{region '#Template'}
	{attribute 'Version' := '5.0.0.0'}
	{attribute 'Tags' := '"LCID": "1031", "Text": "AC, Allgemein, AHU, Startprogramm, Aggregat, Kommandierung"'}
	{attribute 'Tags' := '"LCID": "1033", "Text": "AC, General, AHU, Start program, Aggregate, Command"'}
	{attribute 'Using' := '"Type": "Template", "URI": "E_AC_PlantStep01"'}
	{attribute 'Using' := '"Type": "Template", "URI": "E_BA_AC_OpMod01"'}
	{attribute 'Using' := '"Type": "Template", "URI": "FB_BA_AC_OpModAggBinary"'}
	{attribute 'Using' := '"Type": "Template", "URI": "FB_BA_AC_OpModAggMdlt"'}
	{attribute 'Description' := '"LCID": "1031", "Text": "Kommandierung der Anlage FB_BA_AHU_1st_10"'}
	{attribute 'Description' := '"LCID": "1033", "Text": "Commanding the plant FB_BA_AHU_1st_10"'}
{endregion}

FUNCTION_BLOCK FB_BA_AC_PlantCmd_AHU_1st_10 EXTENDS FB_BA_View
VAR_INPUT
	eOpMode						: E_BA_AC_OpMod01;
	stPriorityEn				: ST_BA_PriorityEn;	
	bDmpOuAOpn					: BOOL;		//	Rückmeldung Aussenluftklappe offen		//	Feedback outside air damper open
	bDmpExhAOpn					: BOOL;		//	Rückmeldung Fortluftklappe offen		//	Feedback exhaust air damper open
	bPreRinse					: BOOL;		//	Vorspülen abgeschlossen					//	Prerinse ready
	bMixADmpAvail				: BOOL;		//	Mischluftsystem vorhanden				//	mixing damper system available	
END_VAR
VAR_OUTPUT
	ePltStp						: E_AC_PlantStep01;	//	Stufen des Anlagenstarts	//	Stages of the plant starts	
	stOuADmp					: ST_BA_Binary;
	stExhADmp					: ST_BA_Binary;
	stSuAFan					: ST_BA_Mdlt;
	stExtAFan					: ST_BA_Mdlt;
	stPreHtr					: ST_BA_Binary;
	stCooler					: ST_BA_Binary;
	stErc						: ST_BA_Binary;
	stTempCtrl					: ST_BA_Mdlt;
	bStepCtrlUp					: BOOL;
	bStepCtrlDown				: BOOL;	
END_VAR
VAR_INPUT CONSTANT
	DmpDlyCls					: FB_BA_AV_Op;
	SuAFanDlyOn					: FB_BA_AV_Op;
	ExtAFanDlyOn				: FB_BA_AV_Op;
	TempCtrlDlyOn				: FB_BA_AV_Op;
	PltStp						: FB_BA_MV_Op;
	
	StepCtrlAgg					: FB_BA_StepCtrlAgg16; //	Schrittsteuerung Aggregate // Step control aggregate	
	

	ErcOpMod					: FB_BA_AC_OpModAggBinary;
	ErcStep						: FB_BA_StepBinary;

	PreHtrOpMod					: FB_BA_AC_OpModAggBinary;
	PreHtrStep					: FB_BA_StepBinary;

	OuADmpOpMod					: FB_BA_AC_OpModAggBinary;
	OuADmpStep					: FB_BA_StepBinary;
	
	SuAFanOpMod					: FB_BA_AC_OpModAggMdlt;
	SuAFanStep					: FB_BA_StepMdlt;	

	ExhADmpOpMod				: FB_BA_AC_OpModAggBinary;
	ExhADmpStep					: FB_BA_StepBinary;
	
	ExtAFanOpMod				: FB_BA_AC_OpModAggMdlt;
	ExtAFanStep					: FB_BA_StepMdlt;	

	CoolerOpMod					: FB_BA_AC_OpModAggBinary;
	CoolerStep					: FB_BA_StepBinary;

	TempCtrlOpMod				: FB_BA_AC_OpModAggMdlt;
	TempCtrlStep				: FB_BA_StepMdlt;	
END_VAR
VAR
	stAgg01						: ST_BA_Step;
	stAgg02						: ST_BA_Step;
	stAgg03						: ST_BA_Step;
	stAgg04						: ST_BA_Step;
	stAgg05						: ST_BA_Step;
	stAgg06						: ST_BA_Step;
	stAgg07						: ST_BA_Step;
	stAgg08						: ST_BA_Step;
	stAgg09						: ST_BA_Step;
	stAgg10						: ST_BA_Step;
	stAgg11						: ST_BA_Step;
	stAgg12						: ST_BA_Step;	
	stAgg13						: ST_BA_Step;	
	stAgg14						: ST_BA_Step;	
	stAgg15						: ST_BA_Step;	
	stAgg16						: ST_BA_Step;	
	
	PltStpMMUX					: FB_BA_MMUX_UDI16;	//	Stufen des Anlagenstarts	//	Stages of the plant starts	
END_VAR

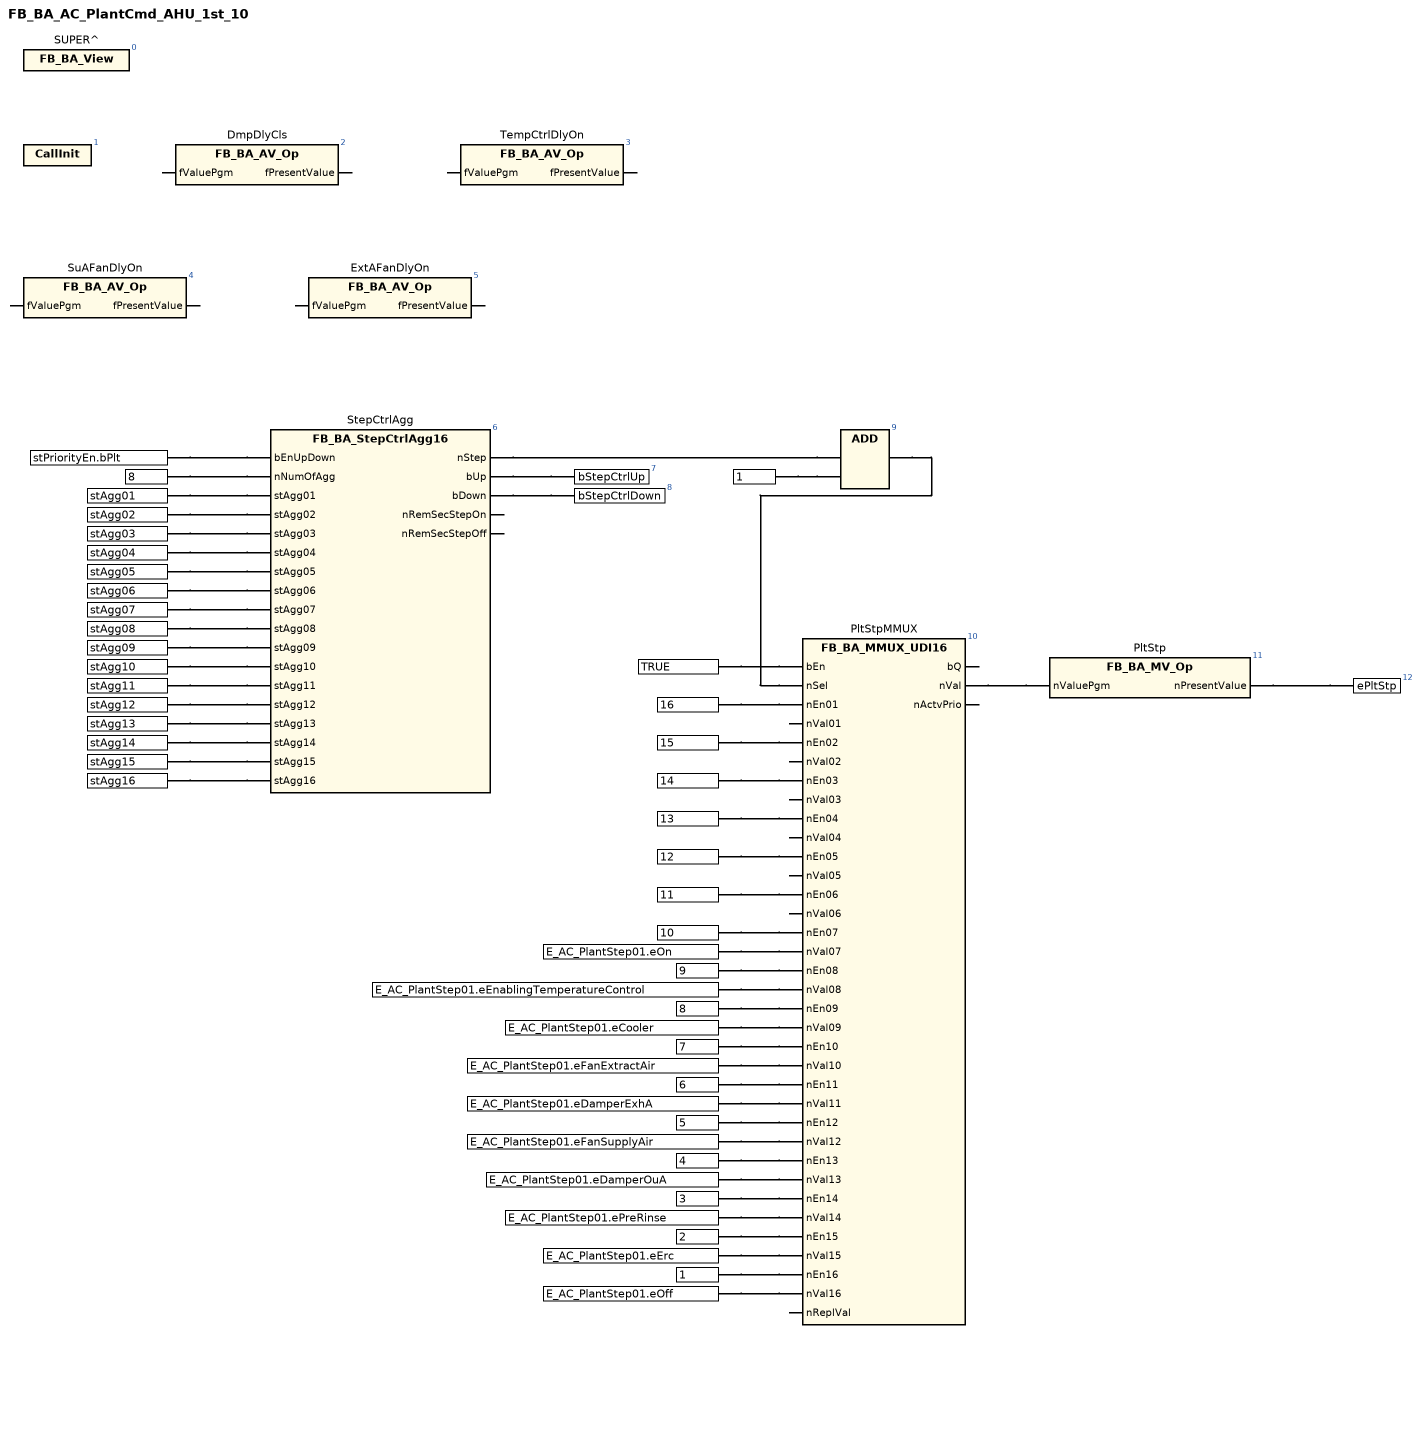
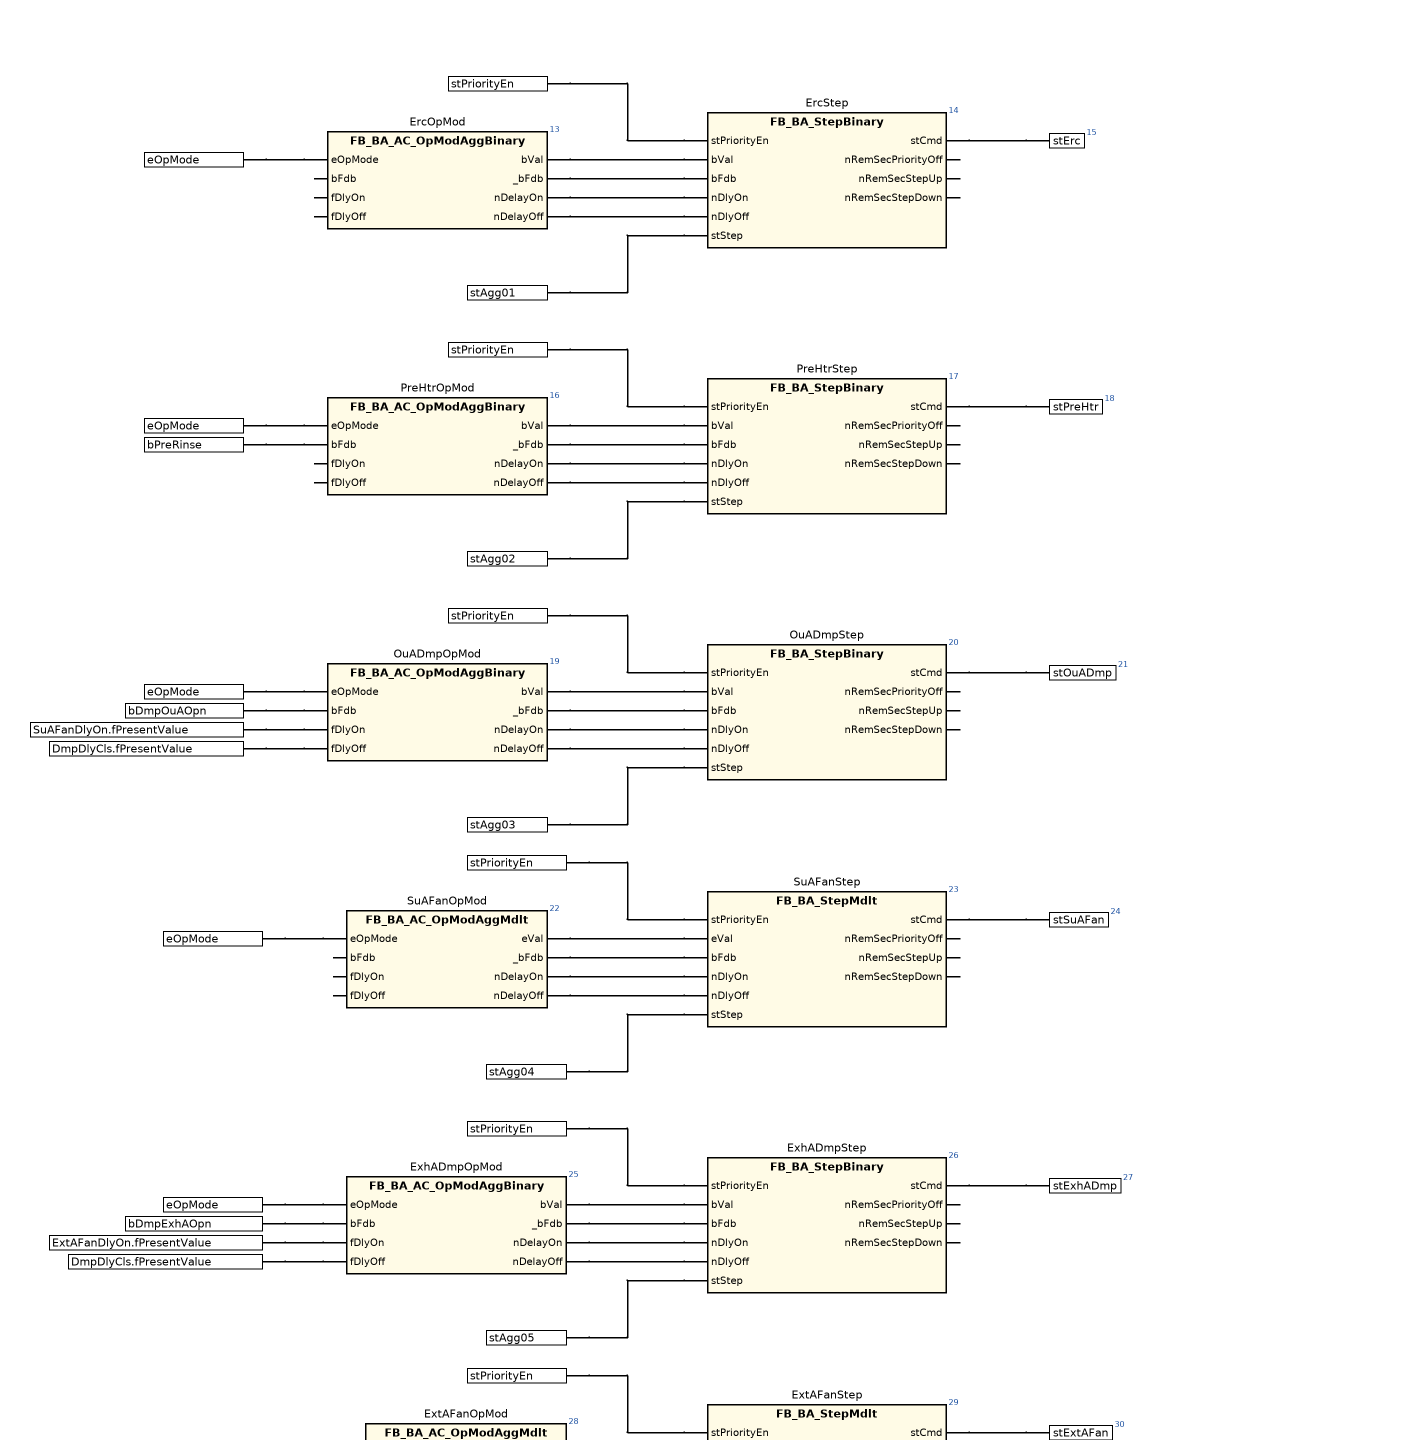
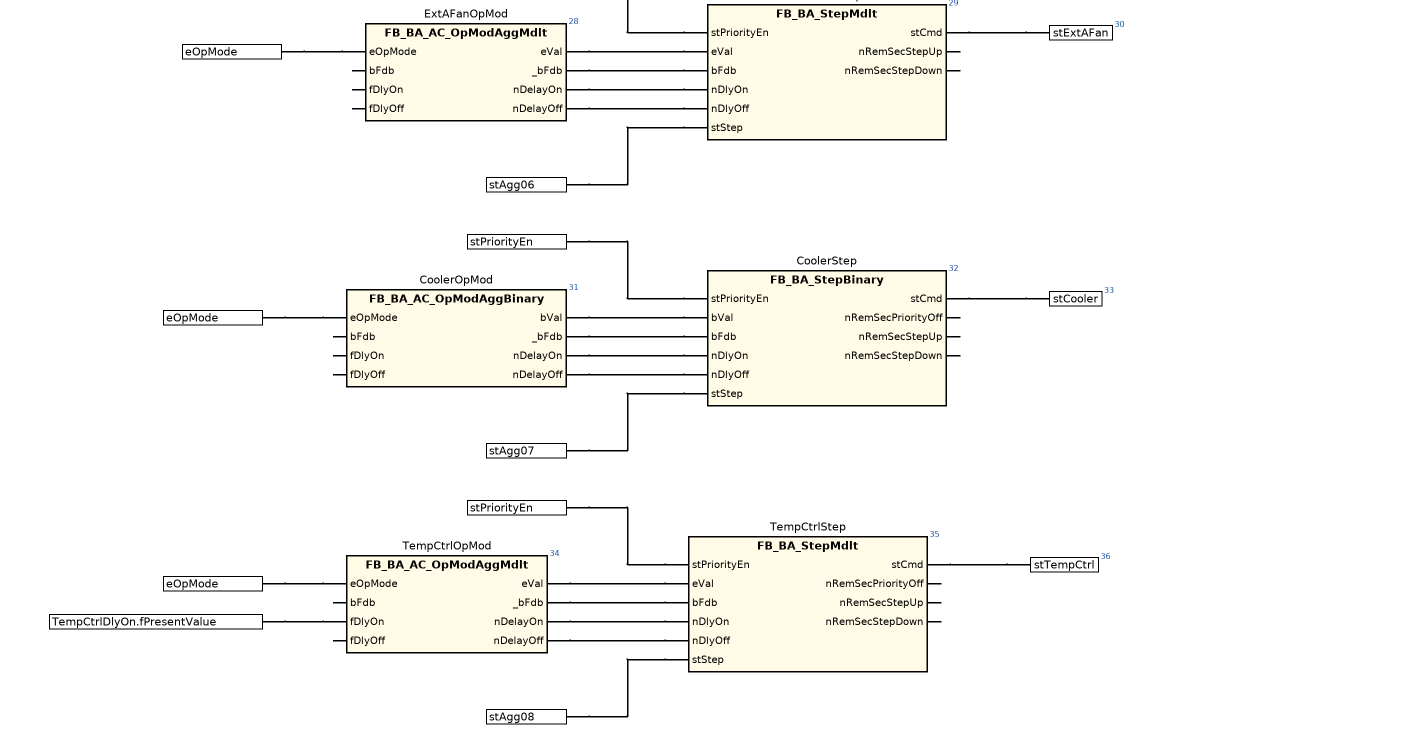
SUPER^(); // FB_BA_View
CallInit();
DmpDlyCls(); // FB_BA_AV_Op
TempCtrlDlyOn(); // FB_BA_AV_Op
SuAFanDlyOn(); // FB_BA_AV_Op
ExtAFanDlyOn(); // FB_BA_AV_Op
StepCtrlAgg(
    bEnUpDown := stPriorityEn.bPlt,
    nNumOfAgg := 8,
    stAgg01 := stAgg01,
    stAgg02 := stAgg02,
    stAgg03 := stAgg03,
    stAgg04 := stAgg04,
    stAgg05 := stAgg05,
    stAgg06 := stAgg06,
    stAgg07 := stAgg07,
    stAgg08 := stAgg08,
    stAgg09 := stAgg09,
    stAgg10 := stAgg10,
    stAgg11 := stAgg11,
    stAgg12 := stAgg12,
    stAgg13 := stAgg13,
    stAgg14 := stAgg14,
    stAgg15 := stAgg15,
    stAgg16 := stAgg16); // FB_BA_StepCtrlAgg16
bStepCtrlUp := StepCtrlAgg.bUp;
bStepCtrlDown := StepCtrlAgg.bDown;
PltStpMMUX(
    bEn := TRUE,
    nSel := StepCtrlAgg.nStep + 1,
    nEn01 := 16,
    nEn02 := 15,
    nEn03 := 14,
    nEn04 := 13,
    nEn05 := 12,
    nEn06 := 11,
    nEn07 := 10,
    nVal07 := E_AC_PlantStep01.eOn,
    nEn08 := 9,
    nVal08 := E_AC_PlantStep01.eEnablingTemperatureControl,
    nEn09 := 8,
    nVal09 := E_AC_PlantStep01.eCooler,
    nEn10 := 7,
    nVal10 := E_AC_PlantStep01.eFanExtractAir,
    nEn11 := 6,
    nVal11 := E_AC_PlantStep01.eDamperExhA,
    nEn12 := 5,
    nVal12 := E_AC_PlantStep01.eFanSupplyAir,
    nEn13 := 4,
    nVal13 := E_AC_PlantStep01.eDamperOuA,
    nEn14 := 3,
    nVal14 := E_AC_PlantStep01.ePreRinse,
    nEn15 := 2,
    nVal15 := E_AC_PlantStep01.eErc,
    nEn16 := 1,
    nVal16 := E_AC_PlantStep01.eOff); // FB_BA_MMUX_UDI16
PltStp(nValuePgm := PltStpMMUX.nVal); // FB_BA_MV_Op
ePltStp := PltStp.nPresentValue;
ErcOpMod(eOpMode := eOpMode); // FB_BA_AC_OpModAggBinary
ErcStep(
    stPriorityEn := stPriorityEn,
    bVal := ErcOpMod.bVal,
    bFdb := ErcOpMod._bFdb,
    nDlyOn := ErcOpMod.nDelayOn,
    nDlyOff := ErcOpMod.nDelayOff,
    stStep := stAgg01); // FB_BA_StepBinary
stErc := ErcStep.stCmd;
PreHtrOpMod(eOpMode := eOpMode, bFdb := bPreRinse); // FB_BA_AC_OpModAggBinary
PreHtrStep(
    stPriorityEn := stPriorityEn,
    bVal := PreHtrOpMod.bVal,
    bFdb := PreHtrOpMod._bFdb,
    nDlyOn := PreHtrOpMod.nDelayOn,
    nDlyOff := PreHtrOpMod.nDelayOff,
    stStep := stAgg02); // FB_BA_StepBinary
stPreHtr := PreHtrStep.stCmd;
OuADmpOpMod(
    eOpMode := eOpMode,
    bFdb := bDmpOuAOpn,
    fDlyOn := SuAFanDlyOn.fPresentValue,
    fDlyOff := DmpDlyCls.fPresentValue); // FB_BA_AC_OpModAggBinary
OuADmpStep(
    stPriorityEn := stPriorityEn,
    bVal := OuADmpOpMod.bVal,
    bFdb := OuADmpOpMod._bFdb,
    nDlyOn := OuADmpOpMod.nDelayOn,
    nDlyOff := OuADmpOpMod.nDelayOff,
    stStep := stAgg03); // FB_BA_StepBinary
stOuADmp := OuADmpStep.stCmd;
SuAFanOpMod(eOpMode := eOpMode); // FB_BA_AC_OpModAggMdlt
SuAFanStep(
    stPriorityEn := stPriorityEn,
    eVal := SuAFanOpMod.eVal,
    bFdb := SuAFanOpMod._bFdb,
    nDlyOn := SuAFanOpMod.nDelayOn,
    nDlyOff := SuAFanOpMod.nDelayOff,
    stStep := stAgg04); // FB_BA_StepMdlt
stSuAFan := SuAFanStep.stCmd;
ExhADmpOpMod(
    eOpMode := eOpMode,
    bFdb := bDmpExhAOpn,
    fDlyOn := ExtAFanDlyOn.fPresentValue,
    fDlyOff := DmpDlyCls.fPresentValue); // FB_BA_AC_OpModAggBinary
ExhADmpStep(
    stPriorityEn := stPriorityEn,
    bVal := ExhADmpOpMod.bVal,
    bFdb := ExhADmpOpMod._bFdb,
    nDlyOn := ExhADmpOpMod.nDelayOn,
    nDlyOff := ExhADmpOpMod.nDelayOff,
    stStep := stAgg05); // FB_BA_StepBinary
stExhADmp := ExhADmpStep.stCmd;
ExtAFanOpMod(eOpMode := eOpMode); // FB_BA_AC_OpModAggMdlt
ExtAFanStep(
    stPriorityEn := stPriorityEn,
    eVal := ExtAFanOpMod.eVal,
    bFdb := ExtAFanOpMod._bFdb,
    nDlyOn := ExtAFanOpMod.nDelayOn,
    nDlyOff := ExtAFanOpMod.nDelayOff,
    stStep := stAgg06); // FB_BA_StepMdlt
stExtAFan := ExtAFanStep.stCmd;
CoolerOpMod(eOpMode := eOpMode); // FB_BA_AC_OpModAggBinary
CoolerStep(
    stPriorityEn := stPriorityEn,
    bVal := CoolerOpMod.bVal,
    bFdb := CoolerOpMod._bFdb,
    nDlyOn := CoolerOpMod.nDelayOn,
    nDlyOff := CoolerOpMod.nDelayOff,
    stStep := stAgg07); // FB_BA_StepBinary
stCooler := CoolerStep.stCmd;
TempCtrlOpMod(eOpMode := eOpMode, fDlyOn := TempCtrlDlyOn.fPresentValue); // FB_BA_AC_OpModAggMdlt
TempCtrlStep(
    stPriorityEn := stPriorityEn,
    eVal := TempCtrlOpMod.eVal,
    bFdb := TempCtrlOpMod._bFdb,
    nDlyOn := TempCtrlOpMod.nDelayOn,
    nDlyOff := TempCtrlOpMod.nDelayOff,
    stStep := stAgg08); // FB_BA_StepMdlt
stTempCtrl := TempCtrlStep.stCmd;

METHOD CallInit
VAR_INPUT
END_VAR
InitErc();
InitPreHtr();

InitOuADmp();
InitSuAFan();

InitExhADmp();
InitExtAFan();

InitCooler();

InitTempCtrl();
END_METHOD

METHOD FB_init : BOOL
VAR_INPUT
	bInitRetains : BOOL; // if TRUE, the retain variables are initialized (warm start / cold start)
	bInCopyCode : BOOL;  // if TRUE, the instance afterwards gets moved into the copy code (online change)
END_VAR
DmpDlyCls.iParent			:= THIS^;
DmpDlyCls.iLabel			:= LblCtl_TimeDelayDampersClose; 	
DmpDlyCls.eUnit				:= E_BA_Unit.eTime_Seconds;  
DmpDlyCls.fValueRm			:= 10;

SuAFanDlyOn.iParent			:= THIS^;
SuAFanDlyOn.iLabel			:= LblCtl_TimeDelaySupplyAirFanOn;   		
SuAFanDlyOn.eUnit			:= E_BA_Unit.eTime_Seconds;  
SuAFanDlyOn.fValueRm		:= 10;

ExtAFanDlyOn.iParent		:= THIS^;
ExtAFanDlyOn.iLabel			:= LblCtl_TimeDelayExtractAirFanOn;   	
ExtAFanDlyOn.eUnit			:= E_BA_Unit.eTime_Seconds;  
ExtAFanDlyOn.fValueRm		:= 10;

TempCtrlDlyOn.iParent		:= THIS^;
TempCtrlDlyOn.iLabel		:= LblCtl_TimeDelayTemperatureSequenceControlOn;   	
TempCtrlDlyOn.eUnit			:= E_BA_Unit.eTime_Seconds;  
TempCtrlDlyOn.fValueRm		:= 5;

PltStp.iParent				:= THIS^;
PltStp.iLabel				:= LblCtl_StagesOfThePlantStartup; 	
PltStp.aStateText[1]		:= txtEvent_Off;
PltStp.aStateText[2]		:= txtEvent_EnergyRecovery;
PltStp.aStateText[3]		:= txtEvent_PreRinse;// or txtEvent_Preheater
PltStp.aStateText[4]		:= txtEvent_DamperOutsideAir;
PltStp.aStateText[5]		:= txtEvent_SupplyAirFan;
PltStp.aStateText[6]		:= txtEvent_DamperExhaustAir;
PltStp.aStateText[7]		:= txtEvent_ExtractAirFan;
PltStp.aStateText[8]		:= txtEvent_Cooler;
PltStp.aStateText[9]		:= txtEvent_Reheater;
PltStp.aStateText[10]		:= txtEvent_MixedAir;
PltStp.aStateText[11]		:= txtEvent_EnableTemperatureControl;
PltStp.aStateText[12]		:= txtEvent_EnableHumidityControl;
PltStp.aStateText[13]		:= txtEvent_On;
END_METHOD

METHOD InitCooler
VAR_INPUT
END_VAR
IF	CoolerOpMod.bInit
THEN	
	CoolerOpMod.bInit := FALSE;
	//////////////////////////////////////////////
	//////////////////////////////////////////////
	//	E_BA_AC_OpMod01.eOff
	CoolerOpMod.arrOpModVal[E_BA_AC_OpMod01.eOff]				:= FALSE;
	CoolerOpMod.arrIgnoreDelayOnVal[E_BA_AC_OpMod01.eOff]		:= TRUE;
	CoolerOpMod.arrIgnoreDelayOffVal[E_BA_AC_OpMod01.eOff]		:= TRUE;
	CoolerOpMod.arrIgnoreFdbVal[E_BA_AC_OpMod01.eOff]			:= TRUE;
	//////////////////////////////////////////////
	//////////////////////////////////////////////
	//	E_BA_AC_OpMod01.eOn
	CoolerOpMod.arrOpModVal[E_BA_AC_OpMod01.eOn]				:= TRUE;
	CoolerOpMod.arrIgnoreDelayOnVal[E_BA_AC_OpMod01.eOn]		:= TRUE;
	CoolerOpMod.arrIgnoreDelayOffVal[E_BA_AC_OpMod01.eOn]		:= TRUE;
	CoolerOpMod.arrIgnoreFdbVal[E_BA_AC_OpMod01.eOn]			:= TRUE;
	//////////////////////////////////////////////
	//////////////////////////////////////////////
	//	E_BA_AC_OpMod01.eEmergency
	CoolerOpMod.arrOpModVal[E_BA_AC_OpMod01.eEmergency]				:= FALSE;
	CoolerOpMod.arrIgnoreDelayOnVal[E_BA_AC_OpMod01.eEmergency]		:= TRUE;
	CoolerOpMod.arrIgnoreDelayOffVal[E_BA_AC_OpMod01.eEmergency]	:= TRUE;
	CoolerOpMod.arrIgnoreFdbVal[E_BA_AC_OpMod01.eEmergency]			:= TRUE;
	//////////////////////////////////////////////
	//////////////////////////////////////////////
	//	E_OpModBA_AC_OpMod01.eFrost
	CoolerOpMod.arrOpModVal[E_BA_AC_OpMod01.eFrost]				:= FALSE;
	CoolerOpMod.arrIgnoreDelayOnVal[E_BA_AC_OpMod01.eFrost]		:= TRUE;
	CoolerOpMod.arrIgnoreDelayOffVal[E_BA_AC_OpMod01.eFrost]	:= TRUE;
	CoolerOpMod.arrIgnoreFdbVal[E_BA_AC_OpMod01.eFrost]			:= TRUE;
	//////////////////////////////////////////////
	//////////////////////////////////////////////
	//	E_BA_AC_OpMod01.eSmokeExtractionProgramm
	CoolerOpMod.arrOpModVal[E_BA_AC_OpMod01.eSmokeExtractionProgram]				:= FALSE;
	CoolerOpMod.arrIgnoreDelayOnVal[E_BA_AC_OpMod01.eSmokeExtractionProgram]		:= TRUE;
	CoolerOpMod.arrIgnoreDelayOffVal[E_BA_AC_OpMod01.eSmokeExtractionProgram]		:= TRUE;
	CoolerOpMod.arrIgnoreFdbVal[E_BA_AC_OpMod01.eSmokeExtractionProgram]			:= TRUE;
	//////////////////////////////////////////////
	//////////////////////////////////////////////
	//	E_BA_AC_OpMod01.eSmokeExtractionSupplyAir
	CoolerOpMod.arrOpModVal[E_BA_AC_OpMod01.eSmokeExtractionSupplyAir]				:= FALSE;
	CoolerOpMod.arrIgnoreDelayOnVal[E_BA_AC_OpMod01.eSmokeExtractionSupplyAir]		:= TRUE;
	CoolerOpMod.arrIgnoreDelayOffVal[E_BA_AC_OpMod01.eSmokeExtractionSupplyAir]		:= TRUE;
	CoolerOpMod.arrIgnoreFdbVal[E_BA_AC_OpMod01.eSmokeExtractionSupplyAir]			:= TRUE;
	//////////////////////////////////////////////
	//////////////////////////////////////////////
	//	E_BA_AC_OpMod01.eSmokeExtractionExhaustAir
	CoolerOpMod.arrOpModVal[E_BA_AC_OpMod01.eSmokeExtractionExhaustAir]				:= FALSE;
	CoolerOpMod.arrIgnoreDelayOnVal[E_BA_AC_OpMod01.eSmokeExtractionExhaustAir]		:= TRUE;
	CoolerOpMod.arrIgnoreDelayOffVal[E_BA_AC_OpMod01.eSmokeExtractionExhaustAir]	:= TRUE;
	CoolerOpMod.arrIgnoreFdbVal[E_BA_AC_OpMod01.eSmokeExtractionExhaustAir]			:= TRUE;
	//////////////////////////////////////////////
	//////////////////////////////////////////////
	//	E_BA_AC_OpMod01.eFire
	CoolerOpMod.arrOpModVal[E_BA_AC_OpMod01.eFire]				:= FALSE;
	CoolerOpMod.arrIgnoreDelayOnVal[E_BA_AC_OpMod01.eFire]		:= TRUE;
	CoolerOpMod.arrIgnoreDelayOffVal[E_BA_AC_OpMod01.eFire]		:= TRUE;
	CoolerOpMod.arrIgnoreFdbVal[E_BA_AC_OpMod01.eFire]			:= TRUE;
	//////////////////////////////////////////////
	//////////////////////////////////////////////
	//	E_BA_AC_OpMod01.eNightCooling
	CoolerOpMod.arrOpModVal[E_BA_AC_OpMod01.eNightCooling]				:= FALSE;
	CoolerOpMod.arrIgnoreDelayOnVal[E_BA_AC_OpMod01.eNightCooling]		:= TRUE;
	CoolerOpMod.arrIgnoreDelayOffVal[E_BA_AC_OpMod01.eNightCooling]		:= TRUE;
	CoolerOpMod.arrIgnoreFdbVal[E_BA_AC_OpMod01.eNightCooling]			:= TRUE;
	//////////////////////////////////////////////
	//////////////////////////////////////////////
	//	E_BA_AC_OpMod01.eCoolDownProtection
	CoolerOpMod.arrOpModVal[E_BA_AC_OpMod01.eCoolDownProtection]				:= FALSE;
	CoolerOpMod.arrIgnoreDelayOnVal[E_BA_AC_OpMod01.eCoolDownProtection]		:= TRUE;
	CoolerOpMod.arrIgnoreDelayOffVal[E_BA_AC_OpMod01.eCoolDownProtection]		:= TRUE;
	CoolerOpMod.arrIgnoreFdbVal[E_BA_AC_OpMod01.eCoolDownProtection]			:= TRUE;
	//////////////////////////////////////////////
	//////////////////////////////////////////////
	//	E_BA_AC_OpMod01.eOverHeatingProtection
	CoolerOpMod.arrOpModVal[E_BA_AC_OpMod01.eOverHeatingProtection]				:= TRUE;
	CoolerOpMod.arrIgnoreDelayOnVal[E_BA_AC_OpMod01.eOverHeatingProtection]		:= TRUE;
	CoolerOpMod.arrIgnoreDelayOffVal[E_BA_AC_OpMod01.eOverHeatingProtection]	:= TRUE;
	CoolerOpMod.arrIgnoreFdbVal[E_BA_AC_OpMod01.eOverHeatingProtection]			:= TRUE;
	//////////////////////////////////////////////
	//////////////////////////////////////////////
	//	E_BA_AC_OpMod01.eAlarm
	CoolerOpMod.arrOpModVal[E_BA_AC_OpMod01.eAlarm]				:= FALSE;
	CoolerOpMod.arrIgnoreDelayOnVal[E_BA_AC_OpMod01.eAlarm]		:= TRUE;
	CoolerOpMod.arrIgnoreDelayOffVal[E_BA_AC_OpMod01.eAlarm]	:= TRUE;
	CoolerOpMod.arrIgnoreFdbVal[E_BA_AC_OpMod01.eAlarm]			:= TRUE;
	//////////////////////////////////////////////
	//////////////////////////////////////////////
	//	E_BA_AC_OpMod01.eForcedVentilation
	CoolerOpMod.arrOpModVal[E_BA_AC_OpMod01.eForcedVentilation]				:= TRUE;
	CoolerOpMod.arrIgnoreDelayOnVal[E_BA_AC_OpMod01.eForcedVentilation]		:= TRUE;
	CoolerOpMod.arrIgnoreDelayOffVal[E_BA_AC_OpMod01.eForcedVentilation]	:= TRUE;
	CoolerOpMod.arrIgnoreFdbVal[E_BA_AC_OpMod01.eForcedVentilation]			:= TRUE;
	//////////////////////////////////////////////
	//////////////////////////////////////////////
	//	E_BA_AC_OpMod01.eCentralSwitchOff
	CoolerOpMod.arrOpModVal[E_BA_AC_OpMod01.eCentralSwitchOff]				:= FALSE;
	CoolerOpMod.arrIgnoreDelayOnVal[E_BA_AC_OpMod01.eCentralSwitchOff]		:= TRUE;
	CoolerOpMod.arrIgnoreDelayOffVal[E_BA_AC_OpMod01.eCentralSwitchOff]		:= TRUE;
	CoolerOpMod.arrIgnoreFdbVal[E_BA_AC_OpMod01.eCentralSwitchOff]			:= TRUE;
	//////////////////////////////////////////////
	//////////////////////////////////////////////
	//	E_BA_AC_OpMod01.eCustomer01
	CoolerOpMod.arrOpModVal[E_BA_AC_OpMod01.eCustomer01]				:= FALSE;
	CoolerOpMod.arrIgnoreDelayOnVal[E_BA_AC_OpMod01.eCustomer01]		:= TRUE;
	CoolerOpMod.arrIgnoreDelayOffVal[E_BA_AC_OpMod01.eCustomer01]		:= TRUE;
	CoolerOpMod.arrIgnoreFdbVal[E_BA_AC_OpMod01.eCustomer01]			:= TRUE;
	//////////////////////////////////////////////
	//////////////////////////////////////////////
	//	E_BA_AC_OpMod01.eCustomer02
	CoolerOpMod.arrOpModVal[E_BA_AC_OpMod01.eCustomer02]				:= FALSE;
	CoolerOpMod.arrIgnoreDelayOnVal[E_BA_AC_OpMod01.eCustomer02]		:= TRUE;
	CoolerOpMod.arrIgnoreDelayOffVal[E_BA_AC_OpMod01.eCustomer02]		:= TRUE;
	CoolerOpMod.arrIgnoreFdbVal[E_BA_AC_OpMod01.eCustomer02]			:= TRUE;
END_IF
END_METHOD

METHOD InitErc
VAR_INPUT
END_VAR
IF	ErcOpMod.bInit
THEN	
	ErcOpMod.bInit := FALSE;
	//////////////////////////////////////////////
	//////////////////////////////////////////////
	//	E_BA_AC_OpMod01.eOff;
	ErcOpMod.arrOpModVal[E_BA_AC_OpMod01.eOff]				:= FALSE;
	ErcOpMod.arrIgnoreDelayOnVal[E_BA_AC_OpMod01.eOff]		:= TRUE;
	ErcOpMod.arrIgnoreDelayOffVal[E_BA_AC_OpMod01.eOff]		:= TRUE;
	ErcOpMod.arrIgnoreFdbVal[E_BA_AC_OpMod01.eOff]			:= TRUE;	
	//////////////////////////////////////////////
	//////////////////////////////////////////////
	//	E_BA_AC_OpMod01.eOn;
	ErcOpMod.arrOpModVal[E_BA_AC_OpMod01.eOn]				:= TRUE;
	ErcOpMod.arrIgnoreDelayOnVal[E_BA_AC_OpMod01.eOn]		:= TRUE;
	ErcOpMod.arrIgnoreDelayOffVal[E_BA_AC_OpMod01.eOn]		:= TRUE;
	ErcOpMod.arrIgnoreFdbVal[E_BA_AC_OpMod01.eOn]			:= TRUE;
	//////////////////////////////////////////////
	//////////////////////////////////////////////
	//	E_BA_AC_OpMod01.eEmergency;
	ErcOpMod.arrOpModVal[E_BA_AC_OpMod01.eEmergency]				:= FALSE;
	ErcOpMod.arrIgnoreDelayOnVal[E_BA_AC_OpMod01.eEmergency]		:= TRUE;
	ErcOpMod.arrIgnoreDelayOffVal[E_BA_AC_OpMod01.eEmergency]		:= TRUE;
	ErcOpMod.arrIgnoreFdbVal[E_BA_AC_OpMod01.eEmergency]			:= TRUE;
	//////////////////////////////////////////////
	//////////////////////////////////////////////
	//	E_BA_AC_OpMod01.eFrost;
	ErcOpMod.arrOpModVal[E_BA_AC_OpMod01.eFrost]				:= FALSE;
	ErcOpMod.arrIgnoreDelayOnVal[E_BA_AC_OpMod01.eFrost]		:= TRUE;
	ErcOpMod.arrIgnoreDelayOffVal[E_BA_AC_OpMod01.eFrost]		:= TRUE;
	ErcOpMod.arrIgnoreFdbVal[E_BA_AC_OpMod01.eFrost]			:= TRUE;
	//////////////////////////////////////////////
	//////////////////////////////////////////////
	//	E_BA_AC_OpMod01.eSmokeExtractionProgramm;
	ErcOpMod.arrOpModVal[E_BA_AC_OpMod01.eSmokeExtractionProgram]				:= FALSE;
	ErcOpMod.arrIgnoreDelayOnVal[E_BA_AC_OpMod01.eSmokeExtractionProgram]		:= TRUE;
	ErcOpMod.arrIgnoreDelayOffVal[E_BA_AC_OpMod01.eSmokeExtractionProgram]		:= TRUE;
	ErcOpMod.arrIgnoreFdbVal[E_BA_AC_OpMod01.eSmokeExtractionProgram]			:= TRUE;
	//////////////////////////////////////////////
	//////////////////////////////////////////////
	//	E_BA_AC_OpMod01.eSmokeExtractionSupplyAir;
	ErcOpMod.arrOpModVal[E_BA_AC_OpMod01.eSmokeExtractionSupplyAir]				:= FALSE;
	ErcOpMod.arrIgnoreDelayOnVal[E_BA_AC_OpMod01.eSmokeExtractionSupplyAir]		:= TRUE;
	ErcOpMod.arrIgnoreDelayOffVal[E_BA_AC_OpMod01.eSmokeExtractionSupplyAir]	:= TRUE;
	ErcOpMod.arrIgnoreFdbVal[E_BA_AC_OpMod01.eSmokeExtractionSupplyAir]			:= TRUE;
	//////////////////////////////////////////////
	//////////////////////////////////////////////
	//	E_BA_AC_OpMod01.eSmokeExtractionExhaustAir;
	ErcOpMod.arrOpModVal[E_BA_AC_OpMod01.eSmokeExtractionExhaustAir]				:= FALSE;
	ErcOpMod.arrIgnoreDelayOnVal[E_BA_AC_OpMod01.eSmokeExtractionExhaustAir]		:= TRUE;
	ErcOpMod.arrIgnoreDelayOffVal[E_BA_AC_OpMod01.eSmokeExtractionExhaustAir]		:= TRUE;
	ErcOpMod.arrIgnoreFdbVal[E_BA_AC_OpMod01.eSmokeExtractionExhaustAir]			:= TRUE;
	//////////////////////////////////////////////
	//////////////////////////////////////////////
	//	E_BA_AC_OpMod01.eFire;
	ErcOpMod.arrOpModVal[E_BA_AC_OpMod01.eFire]				:= FALSE;
	ErcOpMod.arrIgnoreDelayOnVal[E_BA_AC_OpMod01.eFire]		:= TRUE;
	ErcOpMod.arrIgnoreDelayOffVal[E_BA_AC_OpMod01.eFire]	:= TRUE;
	ErcOpMod.arrIgnoreFdbVal[E_BA_AC_OpMod01.eFire]			:= TRUE;
	//////////////////////////////////////////////
	//////////////////////////////////////////////
	//	E_BA_AC_OpMod01.eNightCooling;
	ErcOpMod.arrOpModVal[E_BA_AC_OpMod01.eNightCooling]				:= FALSE;
	ErcOpMod.arrIgnoreDelayOnVal[E_BA_AC_OpMod01.eNightCooling]		:= TRUE;
	ErcOpMod.arrIgnoreDelayOffVal[E_BA_AC_OpMod01.eNightCooling]	:= TRUE;
	ErcOpMod.arrIgnoreFdbVal[E_BA_AC_OpMod01.eNightCooling]			:= TRUE;
	//////////////////////////////////////////////
	//////////////////////////////////////////////
	//	E_BA_AC_OpMod01.eCoolDownProtection;
	ErcOpMod.arrOpModVal[E_BA_AC_OpMod01.eCoolDownProtection]				:= TRUE;
	ErcOpMod.arrIgnoreDelayOnVal[E_BA_AC_OpMod01.eCoolDownProtection]		:= TRUE;
	ErcOpMod.arrIgnoreDelayOffVal[E_BA_AC_OpMod01.eCoolDownProtection]		:= TRUE;
	ErcOpMod.arrIgnoreFdbVal[E_BA_AC_OpMod01.eCoolDownProtection]			:= TRUE;
	//////////////////////////////////////////////
	//////////////////////////////////////////////
	//	E_BA_AC_OpMod01.eOverHeatingProtection;
	ErcOpMod.arrOpModVal[E_BA_AC_OpMod01.eOverHeatingProtection]			:= TRUE;
	ErcOpMod.arrIgnoreDelayOnVal[E_BA_AC_OpMod01.eOverHeatingProtection]	:= TRUE;
	ErcOpMod.arrIgnoreDelayOffVal[E_BA_AC_OpMod01.eOverHeatingProtection]	:= TRUE;
	ErcOpMod.arrIgnoreFdbVal[E_BA_AC_OpMod01.eOverHeatingProtection]		:= TRUE;
	//////////////////////////////////////////////
	//////////////////////////////////////////////
	//	E_BA_AC_OpMod01.eAlarm;
	ErcOpMod.arrOpModVal[E_BA_AC_OpMod01.eAlarm]				:= FALSE;
	ErcOpMod.arrIgnoreDelayOnVal[E_BA_AC_OpMod01.eAlarm]		:= TRUE;
	ErcOpMod.arrIgnoreDelayOffVal[E_BA_AC_OpMod01.eAlarm]		:= TRUE;
	ErcOpMod.arrIgnoreFdbVal[E_BA_AC_OpMod01.eAlarm]			:= TRUE;
	//////////////////////////////////////////////
	//////////////////////////////////////////////
	//	E_BA_AC_OpMod01.eForcedVentilation;
	ErcOpMod.arrOpModVal[E_BA_AC_OpMod01.eForcedVentilation]				:= TRUE;
	ErcOpMod.arrIgnoreDelayOnVal[E_BA_AC_OpMod01.eForcedVentilation]		:= TRUE;
	ErcOpMod.arrIgnoreDelayOffVal[E_BA_AC_OpMod01.eForcedVentilation]		:= TRUE;
	ErcOpMod.arrIgnoreFdbVal[E_BA_AC_OpMod01.eForcedVentilation]			:= TRUE;
	//////////////////////////////////////////////
	//////////////////////////////////////////////
	//	E_BA_AC_OpMod01.eCentralSwitchOff;
	ErcOpMod.arrOpModVal[E_BA_AC_OpMod01.eCentralSwitchOff]				:= FALSE;
	ErcOpMod.arrIgnoreDelayOnVal[E_BA_AC_OpMod01.eCentralSwitchOff]		:= TRUE;
	ErcOpMod.arrIgnoreDelayOffVal[E_BA_AC_OpMod01.eCentralSwitchOff]	:= TRUE;
	ErcOpMod.arrIgnoreFdbVal[E_BA_AC_OpMod01.eCentralSwitchOff]			:= TRUE;
	//////////////////////////////////////////////
	//////////////////////////////////////////////
	//	E_BA_AC_OpMod01.eCustomer01;
	ErcOpMod.arrOpModVal[E_BA_AC_OpMod01.eCustomer01]				:= FALSE;
	ErcOpMod.arrIgnoreDelayOnVal[E_BA_AC_OpMod01.eCustomer01]		:= TRUE;
	ErcOpMod.arrIgnoreDelayOffVal[E_BA_AC_OpMod01.eCustomer01]		:= TRUE;
	ErcOpMod.arrIgnoreFdbVal[E_BA_AC_OpMod01.eCustomer01]			:= TRUE;
	//////////////////////////////////////////////
	//////////////////////////////////////////////
	//	E_BA_AC_OpMod01.eCustomer02;
	ErcOpMod.arrOpModVal[E_BA_AC_OpMod01.eCustomer02]				:= FALSE;
	ErcOpMod.arrIgnoreDelayOnVal[E_BA_AC_OpMod01.eCustomer02]		:= TRUE;
	ErcOpMod.arrIgnoreDelayOffVal[E_BA_AC_OpMod01.eCustomer02]		:= TRUE;
	ErcOpMod.arrIgnoreFdbVal[E_BA_AC_OpMod01.eCustomer02]			:= TRUE;
END_IF
END_METHOD

METHOD InitExhADmp
VAR_INPUT
END_VAR
IF	ExhADmpOpMod.bInit
THEN	
	ExhADmpOpMod.bInit := FALSE;
	//////////////////////////////////////////////
	//////////////////////////////////////////////
	//	E_BA_AC_OpMod01.eOff
	ExhADmpOpMod.arrOpModVal[E_BA_AC_OpMod01.eOff]				:= FALSE;
	ExhADmpOpMod.arrIgnoreDelayOnVal[E_BA_AC_OpMod01.eOff]		:= TRUE;
	ExhADmpOpMod.arrIgnoreDelayOffVal[E_BA_AC_OpMod01.eOff]		:= FALSE;
	ExhADmpOpMod.arrIgnoreFdbVal[E_BA_AC_OpMod01.eOff]			:= TRUE;
	//////////////////////////////////////////////
	//////////////////////////////////////////////
	//	E_BA_AC_OpMod01.eOn;
	ExhADmpOpMod.arrOpModVal[E_BA_AC_OpMod01.eOn]				:= TRUE;
	ExhADmpOpMod.arrIgnoreDelayOnVal[E_BA_AC_OpMod01.eOn]		:= TRUE;
	ExhADmpOpMod.arrIgnoreDelayOffVal[E_BA_AC_OpMod01.eOn]		:= TRUE;
	ExhADmpOpMod.arrIgnoreFdbVal[E_BA_AC_OpMod01.eOn]			:= FALSE;
	//////////////////////////////////////////////
	//////////////////////////////////////////////
	//	E_BA_AC_OpMod01.eEmergency;
	ExhADmpOpMod.arrOpModVal[E_BA_AC_OpMod01.eEmergency]				:= FALSE;
	ExhADmpOpMod.arrIgnoreDelayOnVal[E_BA_AC_OpMod01.eEmergency]		:= TRUE;
	ExhADmpOpMod.arrIgnoreDelayOffVal[E_BA_AC_OpMod01.eEmergency]		:= TRUE;
	ExhADmpOpMod.arrIgnoreFdbVal[E_BA_AC_OpMod01.eEmergency]			:= TRUE;
	//////////////////////////////////////////////
	//////////////////////////////////////////////
	//	E_BA_AC_OpMod01.eFrost;
	ExhADmpOpMod.arrOpModVal[E_BA_AC_OpMod01.eFrost]				:= FALSE;
	ExhADmpOpMod.arrIgnoreDelayOnVal[E_BA_AC_OpMod01.eFrost]		:= TRUE;
	ExhADmpOpMod.arrIgnoreDelayOffVal[E_BA_AC_OpMod01.eFrost]		:= FALSE;
	ExhADmpOpMod.arrIgnoreFdbVal[E_BA_AC_OpMod01.eFrost]			:= TRUE;
	//////////////////////////////////////////////
	//////////////////////////////////////////////
	//	E_BA_AC_OpMod01.eSmokeExtractionProgramm;
	ExhADmpOpMod.arrOpModVal[E_BA_AC_OpMod01.eSmokeExtractionProgram]				:= TRUE;
	ExhADmpOpMod.arrIgnoreDelayOnVal[E_BA_AC_OpMod01.eSmokeExtractionProgram]		:= TRUE;
	ExhADmpOpMod.arrIgnoreDelayOffVal[E_BA_AC_OpMod01.eSmokeExtractionProgram]		:= TRUE;
	ExhADmpOpMod.arrIgnoreFdbVal[E_BA_AC_OpMod01.eSmokeExtractionProgram]			:= TRUE;
	//////////////////////////////////////////////
	//////////////////////////////////////////////
	//	E_BA_AC_OpMod01.eSmokeExtractionSupplyAir;
	ExhADmpOpMod.arrOpModVal[E_BA_AC_OpMod01.eSmokeExtractionSupplyAir]				:= FALSE;
	ExhADmpOpMod.arrIgnoreDelayOnVal[E_BA_AC_OpMod01.eSmokeExtractionSupplyAir]		:= TRUE;
	ExhADmpOpMod.arrIgnoreDelayOffVal[E_BA_AC_OpMod01.eSmokeExtractionSupplyAir]	:= FALSE;
	ExhADmpOpMod.arrIgnoreFdbVal[E_BA_AC_OpMod01.eSmokeExtractionSupplyAir]			:= TRUE;
	//////////////////////////////////////////////
	//////////////////////////////////////////////
	//	E_BA_AC_OpMod01.eSmokeExtractionExhaustAir;
	ExhADmpOpMod.arrOpModVal[E_BA_AC_OpMod01.eSmokeExtractionExhaustAir]				:= TRUE;
	ExhADmpOpMod.arrIgnoreDelayOnVal[E_BA_AC_OpMod01.eSmokeExtractionExhaustAir]		:= TRUE;
	ExhADmpOpMod.arrIgnoreDelayOffVal[E_BA_AC_OpMod01.eSmokeExtractionExhaustAir]		:= TRUE;
	ExhADmpOpMod.arrIgnoreFdbVal[E_BA_AC_OpMod01.eSmokeExtractionExhaustAir]			:= TRUE;
	//////////////////////////////////////////////
	//////////////////////////////////////////////
	//	E_BA_AC_OpMod01.eFire;
	ExhADmpOpMod.arrOpModVal[E_BA_AC_OpMod01.eFire]				:= FALSE;
	ExhADmpOpMod.arrIgnoreDelayOnVal[E_BA_AC_OpMod01.eFire]		:= TRUE;
	ExhADmpOpMod.arrIgnoreDelayOffVal[E_BA_AC_OpMod01.eFire]	:= TRUE;
	ExhADmpOpMod.arrIgnoreFdbVal[E_BA_AC_OpMod01.eFire]			:= TRUE;
	//////////////////////////////////////////////
	//////////////////////////////////////////////
	//	E_BA_AC_OpMod01.eNightCooling;
	ExhADmpOpMod.arrOpModVal[E_BA_AC_OpMod01.eNightCooling]				:= TRUE;
	ExhADmpOpMod.arrIgnoreDelayOnVal[E_BA_AC_OpMod01.eNightCooling]		:= TRUE;
	ExhADmpOpMod.arrIgnoreDelayOffVal[E_BA_AC_OpMod01.eNightCooling]	:= TRUE;
	ExhADmpOpMod.arrIgnoreFdbVal[E_BA_AC_OpMod01.eNightCooling]			:= FALSE;
	//////////////////////////////////////////////
	//////////////////////////////////////////////
	//	E_BA_AC_OpMod01.eCoolDownProtection;
	ExhADmpOpMod.arrOpModVal[E_BA_AC_OpMod01.eCoolDownProtection]				:= TRUE;
	ExhADmpOpMod.arrIgnoreDelayOnVal[E_BA_AC_OpMod01.eCoolDownProtection]		:= TRUE;
	ExhADmpOpMod.arrIgnoreDelayOffVal[E_BA_AC_OpMod01.eCoolDownProtection]		:= TRUE;
	ExhADmpOpMod.arrIgnoreFdbVal[E_BA_AC_OpMod01.eCoolDownProtection]			:= FALSE;
	//////////////////////////////////////////////
	//////////////////////////////////////////////
	//	E_BA_AC_OpMod01.eOverHeatingProtection;
	ExhADmpOpMod.arrOpModVal[E_BA_AC_OpMod01.eOverHeatingProtection]				:= TRUE;
	ExhADmpOpMod.arrIgnoreDelayOnVal[E_BA_AC_OpMod01.eOverHeatingProtection]		:= TRUE;
	ExhADmpOpMod.arrIgnoreDelayOffVal[E_BA_AC_OpMod01.eOverHeatingProtection]		:= TRUE;
	ExhADmpOpMod.arrIgnoreFdbVal[E_BA_AC_OpMod01.eOverHeatingProtection]			:= FALSE;
	//////////////////////////////////////////////
	//////////////////////////////////////////////
	//	E_BA_AC_OpMod01.eAlarm;
	ExhADmpOpMod.arrOpModVal[E_BA_AC_OpMod01.eAlarm]				:= FALSE;
	ExhADmpOpMod.arrIgnoreDelayOnVal[E_BA_AC_OpMod01.eAlarm]		:= TRUE;
	ExhADmpOpMod.arrIgnoreDelayOffVal[E_BA_AC_OpMod01.eAlarm]		:= FALSE;
	ExhADmpOpMod.arrIgnoreFdbVal[E_BA_AC_OpMod01.eAlarm]			:= TRUE;
	//////////////////////////////////////////////
	//////////////////////////////////////////////
	//	E_BA_AC_OpMod01.eForcedVentilation;
	ExhADmpOpMod.arrOpModVal[E_BA_AC_OpMod01.eForcedVentilation]				:= TRUE;
	ExhADmpOpMod.arrIgnoreDelayOnVal[E_BA_AC_OpMod01.eForcedVentilation]		:= TRUE;
	ExhADmpOpMod.arrIgnoreDelayOffVal[E_BA_AC_OpMod01.eForcedVentilation]		:= TRUE;
	ExhADmpOpMod.arrIgnoreFdbVal[E_BA_AC_OpMod01.eForcedVentilation]			:= FALSE;
	//////////////////////////////////////////////
	//////////////////////////////////////////////
	//	E_BA_AC_OpMod01.eCentralSwitchOff;
	ExhADmpOpMod.arrOpModVal[E_BA_AC_OpMod01.eCentralSwitchOff]				:= FALSE;
	ExhADmpOpMod.arrIgnoreDelayOnVal[E_BA_AC_OpMod01.eCentralSwitchOff]		:= TRUE;
	ExhADmpOpMod.arrIgnoreDelayOffVal[E_BA_AC_OpMod01.eCentralSwitchOff]	:= FALSE;
	ExhADmpOpMod.arrIgnoreFdbVal[E_BA_AC_OpMod01.eCentralSwitchOff]			:= TRUE;
	//////////////////////////////////////////////
	//////////////////////////////////////////////
	//	E_BA_AC_OpMod01.eCustomer01;
	ExhADmpOpMod.arrOpModVal[E_BA_AC_OpMod01.eCustomer01]				:= FALSE;
	ExhADmpOpMod.arrIgnoreDelayOnVal[E_BA_AC_OpMod01.eCustomer01]		:= TRUE;
	ExhADmpOpMod.arrIgnoreDelayOffVal[E_BA_AC_OpMod01.eCustomer01]		:= FALSE;
	ExhADmpOpMod.arrIgnoreFdbVal[E_BA_AC_OpMod01.eCustomer01]			:= TRUE;
	//////////////////////////////////////////////
	//////////////////////////////////////////////
	//	E_BA_AC_OpMod01.eCustomer02;
	ExhADmpOpMod.arrOpModVal[E_BA_AC_OpMod01.eCustomer02]				:= FALSE;
	ExhADmpOpMod.arrIgnoreDelayOnVal[E_BA_AC_OpMod01.eCustomer02]		:= TRUE;
	ExhADmpOpMod.arrIgnoreDelayOffVal[E_BA_AC_OpMod01.eCustomer02]		:= FALSE;
	ExhADmpOpMod.arrIgnoreFdbVal[E_BA_AC_OpMod01.eCustomer02]			:= TRUE;
END_IF
END_METHOD

METHOD InitExtAFan
VAR_INPUT
END_VAR
IF	ExtAFanOpMod.bInit
THEN	
	ExtAFanOpMod.bInit := FALSE;
	//////////////////////////////////////////////
	//////////////////////////////////////////////
	//	E_BA_AC_OpMod01.eOff;
	ExtAFanOpMod.arrOpModVal[E_BA_AC_OpMod01.eOff]				:= E_BA_Mdlt.eOff;
	ExtAFanOpMod.arrIgnoreDelayOnVal[E_BA_AC_OpMod01.eOff]		:= TRUE;
	ExtAFanOpMod.arrIgnoreDelayOffVal[E_BA_AC_OpMod01.eOff]		:= TRUE;
	ExtAFanOpMod.arrIgnoreFdbVal[E_BA_AC_OpMod01.eOff]			:= TRUE;
	//////////////////////////////////////////////
	//////////////////////////////////////////////
	//	E_BA_AC_OpMod01.eOn;
	ExtAFanOpMod.arrOpModVal[E_BA_AC_OpMod01.eOn]				:= E_BA_Mdlt.eOn;
	ExtAFanOpMod.arrIgnoreDelayOnVal[E_BA_AC_OpMod01.eOn]		:= FALSE;
	ExtAFanOpMod.arrIgnoreDelayOffVal[E_BA_AC_OpMod01.eOn]		:= TRUE;
	ExtAFanOpMod.arrIgnoreFdbVal[E_BA_AC_OpMod01.eOn]			:= TRUE;
	//////////////////////////////////////////////
	//////////////////////////////////////////////
	//	E_BA_AC_OpMod01.eEmergency;
	ExtAFanOpMod.arrOpModVal[E_BA_AC_OpMod01.eEmergency]				:= E_BA_Mdlt.eOff;
	ExtAFanOpMod.arrIgnoreDelayOnVal[E_BA_AC_OpMod01.eEmergency]		:= TRUE;
	ExtAFanOpMod.arrIgnoreDelayOffVal[E_BA_AC_OpMod01.eEmergency]		:= TRUE;
	ExtAFanOpMod.arrIgnoreFdbVal[E_BA_AC_OpMod01.eEmergency]			:= TRUE;
	//////////////////////////////////////////////
	//////////////////////////////////////////////
	//	E_BA_AC_OpMod01.eFrost;
	ExtAFanOpMod.arrOpModVal[E_BA_AC_OpMod01.eFrost]				:= E_BA_Mdlt.eOff;
	ExtAFanOpMod.arrIgnoreDelayOnVal[E_BA_AC_OpMod01.eFrost]		:= TRUE;
	ExtAFanOpMod.arrIgnoreDelayOffVal[E_BA_AC_OpMod01.eFrost]		:= TRUE;
	ExtAFanOpMod.arrIgnoreFdbVal[E_BA_AC_OpMod01.eFrost]			:= TRUE;
	//////////////////////////////////////////////
	//////////////////////////////////////////////
	//	E_BA_AC_OpMod01.eSmokeExtractionProgramm;
	ExtAFanOpMod.arrOpModVal[E_BA_AC_OpMod01.eSmokeExtractionProgram]				:= E_BA_Mdlt.eOn;
	ExtAFanOpMod.arrIgnoreDelayOnVal[E_BA_AC_OpMod01.eSmokeExtractionProgram]		:= TRUE;
	ExtAFanOpMod.arrIgnoreDelayOffVal[E_BA_AC_OpMod01.eSmokeExtractionProgram]		:= TRUE;
	ExtAFanOpMod.arrIgnoreFdbVal[E_BA_AC_OpMod01.eSmokeExtractionProgram]			:= TRUE;
	//////////////////////////////////////////////
	//////////////////////////////////////////////
	//	E_BA_AC_OpMod01.eSmokeExtractionSupplyAir;
	ExtAFanOpMod.arrOpModVal[E_BA_AC_OpMod01.eSmokeExtractionSupplyAir]				:= E_BA_Mdlt.eOff;
	ExtAFanOpMod.arrIgnoreDelayOnVal[E_BA_AC_OpMod01.eSmokeExtractionSupplyAir]		:= TRUE;
	ExtAFanOpMod.arrIgnoreDelayOffVal[E_BA_AC_OpMod01.eSmokeExtractionSupplyAir]	:= TRUE;
	ExtAFanOpMod.arrIgnoreFdbVal[E_BA_AC_OpMod01.eSmokeExtractionSupplyAir]			:= TRUE;
	//////////////////////////////////////////////
	//////////////////////////////////////////////
	//	E_BA_AC_OpMod01.eSmokeExtractionExhaustAir;
	ExtAFanOpMod.arrOpModVal[E_BA_AC_OpMod01.eSmokeExtractionExhaustAir]				:= E_BA_Mdlt.eOn;
	ExtAFanOpMod.arrIgnoreDelayOnVal[E_BA_AC_OpMod01.eSmokeExtractionExhaustAir]		:= TRUE;
	ExtAFanOpMod.arrIgnoreDelayOffVal[E_BA_AC_OpMod01.eSmokeExtractionExhaustAir]		:= TRUE;
	ExtAFanOpMod.arrIgnoreFdbVal[E_BA_AC_OpMod01.eSmokeExtractionExhaustAir]			:= TRUE;
	//////////////////////////////////////////////
	//////////////////////////////////////////////
	//	E_BA_AC_OpMod01.eFire;
	ExtAFanOpMod.arrOpModVal[E_BA_AC_OpMod01.eFire]				:= E_BA_Mdlt.eOff;
	ExtAFanOpMod.arrIgnoreDelayOnVal[E_BA_AC_OpMod01.eFire]		:= TRUE;
	ExtAFanOpMod.arrIgnoreDelayOffVal[E_BA_AC_OpMod01.eFire]	:= TRUE;
	ExtAFanOpMod.arrIgnoreFdbVal[E_BA_AC_OpMod01.eFire]			:= TRUE;
	//////////////////////////////////////////////
	//////////////////////////////////////////////
	//	E_BA_AC_OpMod01.eNightCooling;
	ExtAFanOpMod.arrOpModVal[E_BA_AC_OpMod01.eNightCooling]				:= E_BA_Mdlt.eOn;
	ExtAFanOpMod.arrIgnoreDelayOnVal[E_BA_AC_OpMod01.eNightCooling]		:= TRUE;
	ExtAFanOpMod.arrIgnoreDelayOffVal[E_BA_AC_OpMod01.eNightCooling]	:= TRUE;
	ExtAFanOpMod.arrIgnoreFdbVal[E_BA_AC_OpMod01.eNightCooling]			:= TRUE;
	//////////////////////////////////////////////
	//////////////////////////////////////////////
	//	E_BA_AC_OpMod01.eCoolDownProtection;
	ExtAFanOpMod.arrOpModVal[E_BA_AC_OpMod01.eCoolDownProtection]				:= E_BA_Mdlt.eOn;
	ExtAFanOpMod.arrIgnoreDelayOnVal[E_BA_AC_OpMod01.eCoolDownProtection]		:= TRUE;
	ExtAFanOpMod.arrIgnoreDelayOffVal[E_BA_AC_OpMod01.eCoolDownProtection]		:= TRUE;
	ExtAFanOpMod.arrIgnoreFdbVal[E_BA_AC_OpMod01.eCoolDownProtection]			:= TRUE;
	//////////////////////////////////////////////
	//////////////////////////////////////////////
	//	E_BA_AC_OpMod01.eOverHeatingProtection;
	ExtAFanOpMod.arrOpModVal[E_BA_AC_OpMod01.eOverHeatingProtection]				:= E_BA_Mdlt.eOn;
	ExtAFanOpMod.arrIgnoreDelayOnVal[E_BA_AC_OpMod01.eOverHeatingProtection]		:= TRUE;
	ExtAFanOpMod.arrIgnoreDelayOffVal[E_BA_AC_OpMod01.eOverHeatingProtection]		:= TRUE;
	ExtAFanOpMod.arrIgnoreFdbVal[E_BA_AC_OpMod01.eOverHeatingProtection]			:= TRUE;
	//////////////////////////////////////////////
	//////////////////////////////////////////////
	//	E_BA_AC_OpMod01.eAlarm;
	ExtAFanOpMod.arrOpModVal[E_BA_AC_OpMod01.eAlarm]				:= E_BA_Mdlt.eOff;
	ExtAFanOpMod.arrIgnoreDelayOnVal[E_BA_AC_OpMod01.eAlarm]		:= TRUE;
	ExtAFanOpMod.arrIgnoreDelayOffVal[E_BA_AC_OpMod01.eAlarm]		:= TRUE;
	ExtAFanOpMod.arrIgnoreFdbVal[E_BA_AC_OpMod01.eAlarm]			:= TRUE;
	//////////////////////////////////////////////
	//////////////////////////////////////////////
	//	E_BA_AC_OpMod01.eForcedVentilation;
	ExtAFanOpMod.arrOpModVal[E_BA_AC_OpMod01.eForcedVentilation]				:= E_BA_Mdlt.eOn;
	ExtAFanOpMod.arrIgnoreDelayOnVal[E_BA_AC_OpMod01.eForcedVentilation]		:= TRUE;
	ExtAFanOpMod.arrIgnoreDelayOffVal[E_BA_AC_OpMod01.eForcedVentilation]		:= TRUE;
	ExtAFanOpMod.arrIgnoreFdbVal[E_BA_AC_OpMod01.eForcedVentilation]			:= TRUE;
	//////////////////////////////////////////////
	//////////////////////////////////////////////
	//	E_BA_AC_OpMod01.eCentralSwitchOff;
	ExtAFanOpMod.arrOpModVal[E_BA_AC_OpMod01.eCentralSwitchOff]				:= E_BA_Mdlt.eOff;
	ExtAFanOpMod.arrIgnoreDelayOnVal[E_BA_AC_OpMod01.eCentralSwitchOff]		:= TRUE;
	ExtAFanOpMod.arrIgnoreDelayOffVal[E_BA_AC_OpMod01.eCentralSwitchOff]	:= TRUE;
	ExtAFanOpMod.arrIgnoreFdbVal[E_BA_AC_OpMod01.eCentralSwitchOff]			:= TRUE;
	//////////////////////////////////////////////
	//////////////////////////////////////////////
	//	E_BA_AC_OpMod01.eCustomer01;
	ExtAFanOpMod.arrOpModVal[E_BA_AC_OpMod01.eCustomer01]				:= E_BA_Mdlt.eOff;
	ExtAFanOpMod.arrIgnoreDelayOnVal[E_BA_AC_OpMod01.eCustomer01]		:= TRUE;
	ExtAFanOpMod.arrIgnoreDelayOffVal[E_BA_AC_OpMod01.eCustomer01]		:= TRUE;
	ExtAFanOpMod.arrIgnoreFdbVal[E_BA_AC_OpMod01.eCustomer01]			:= TRUE;
	//////////////////////////////////////////////
	//////////////////////////////////////////////
	//	E_BA_AC_OpMod01.eCustomer02;
	ExtAFanOpMod.arrOpModVal[E_BA_AC_OpMod01.eCustomer02]				:= E_BA_Mdlt.eOff;
	ExtAFanOpMod.arrIgnoreDelayOnVal[E_BA_AC_OpMod01.eCustomer02]		:= TRUE;
	ExtAFanOpMod.arrIgnoreDelayOffVal[E_BA_AC_OpMod01.eCustomer02]		:= TRUE;
	ExtAFanOpMod.arrIgnoreFdbVal[E_BA_AC_OpMod01.eCustomer02]			:= TRUE;
END_IF
END_METHOD

METHOD InitOuADmp
VAR_INPUT
END_VAR
IF	OuADmpOpMod.bInit
THEN	
	OuADmpOpMod.bInit := FALSE;
	//////////////////////////////////////////////
	//////////////////////////////////////////////
	//	E_BA_AC_OpMod01.eOff;
	OuADmpOpMod.arrOpModVal[E_BA_AC_OpMod01.eOff]				:= FALSE;
	OuADmpOpMod.arrIgnoreDelayOnVal[E_BA_AC_OpMod01.eOff]		:= TRUE;
	OuADmpOpMod.arrIgnoreDelayOffVal[E_BA_AC_OpMod01.eOff]		:= FALSE;
	OuADmpOpMod.arrIgnoreFdbVal[E_BA_AC_OpMod01.eOff]			:= TRUE;
	//////////////////////////////////////////////
	//////////////////////////////////////////////
	//	E_BA_AC_OpMod01.eOn;
	OuADmpOpMod.arrOpModVal[E_BA_AC_OpMod01.eOn]				:= TRUE;
	OuADmpOpMod.arrIgnoreDelayOnVal[E_BA_AC_OpMod01.eOn]		:= TRUE;
	OuADmpOpMod.arrIgnoreDelayOffVal[E_BA_AC_OpMod01.eOn]	:= TRUE;
	OuADmpOpMod.arrIgnoreFdbVal[E_BA_AC_OpMod01.eOn]			:= FALSE;
	//////////////////////////////////////////////
	//////////////////////////////////////////////	
	//	E_BA_AC_OpMod01.eEmergency;
	OuADmpOpMod.arrOpModVal[E_BA_AC_OpMod01.eEmergency]				:= FALSE;
	OuADmpOpMod.arrIgnoreDelayOnVal[E_BA_AC_OpMod01.eEmergency]		:= TRUE;
	OuADmpOpMod.arrIgnoreDelayOffVal[E_BA_AC_OpMod01.eEmergency]		:= FALSE;
	OuADmpOpMod.arrIgnoreFdbVal[E_BA_AC_OpMod01.eEmergency]			:= TRUE;
	//////////////////////////////////////////////
	//////////////////////////////////////////////
	//	E_BA_AC_OpMod01.eFrost;
	OuADmpOpMod.arrOpModVal[E_BA_AC_OpMod01.eFrost]				:= FALSE;
	OuADmpOpMod.arrIgnoreDelayOnVal[E_BA_AC_OpMod01.eFrost]		:= TRUE;
	OuADmpOpMod.arrIgnoreDelayOffVal[E_BA_AC_OpMod01.eFrost]		:= FALSE;
	OuADmpOpMod.arrIgnoreFdbVal[E_BA_AC_OpMod01.eFrost]			:= TRUE;
	//////////////////////////////////////////////
	//////////////////////////////////////////////
	//	E_BA_AC_OpMod01.eSmokeExtractionProgram;
	OuADmpOpMod.arrOpModVal[E_BA_AC_OpMod01.eSmokeExtractionProgram]				:= TRUE;
	OuADmpOpMod.arrIgnoreDelayOnVal[E_BA_AC_OpMod01.eSmokeExtractionProgram]		:= TRUE;
	OuADmpOpMod.arrIgnoreDelayOffVal[E_BA_AC_OpMod01.eSmokeExtractionProgram]		:= TRUE;
	OuADmpOpMod.arrIgnoreFdbVal[E_BA_AC_OpMod01.eSmokeExtractionProgram]			:= FALSE;
	//////////////////////////////////////////////
	//////////////////////////////////////////////
	//	E_BA_AC_OpMod01.eSmokeExtractionSupplyAir;
	OuADmpOpMod.arrOpModVal[E_BA_AC_OpMod01.eSmokeExtractionSupplyAir]				:= TRUE;
	OuADmpOpMod.arrIgnoreDelayOnVal[E_BA_AC_OpMod01.eSmokeExtractionSupplyAir]		:= TRUE;
	OuADmpOpMod.arrIgnoreDelayOffVal[E_BA_AC_OpMod01.eSmokeExtractionSupplyAir]		:= TRUE;
	OuADmpOpMod.arrIgnoreFdbVal[E_BA_AC_OpMod01.eSmokeExtractionSupplyAir]			:= FALSE;
	//////////////////////////////////////////////
	//////////////////////////////////////////////	
	//	E_BA_AC_OpMod01.eSmokeExtractionExhaustAir;
	OuADmpOpMod.arrOpModVal[E_BA_AC_OpMod01.eSmokeExtractionExhaustAir]				:= FALSE;
	OuADmpOpMod.arrIgnoreDelayOnVal[E_BA_AC_OpMod01.eSmokeExtractionExhaustAir]		:= TRUE;
	OuADmpOpMod.arrIgnoreDelayOffVal[E_BA_AC_OpMod01.eSmokeExtractionExhaustAir]		:= FALSE;
	OuADmpOpMod.arrIgnoreFdbVal[E_BA_AC_OpMod01.eSmokeExtractionExhaustAir]			:= TRUE;
	//////////////////////////////////////////////
	//////////////////////////////////////////////
	//	E_BA_AC_OpMod01.eFire;
	OuADmpOpMod.arrOpModVal[E_BA_AC_OpMod01.eFire]				:= FALSE;
	OuADmpOpMod.arrIgnoreDelayOnVal[E_BA_AC_OpMod01.eFire]		:= TRUE;
	OuADmpOpMod.arrIgnoreDelayOffVal[E_BA_AC_OpMod01.eFire]		:= TRUE;
	OuADmpOpMod.arrIgnoreFdbVal[E_BA_AC_OpMod01.eFire]			:= TRUE;
	//////////////////////////////////////////////
	//////////////////////////////////////////////
	//	E_BA_AC_OpMod01.eNightCooling;
	OuADmpOpMod.arrOpModVal[E_BA_AC_OpMod01.eNightCooling]				:= TRUE;
	OuADmpOpMod.arrIgnoreDelayOnVal[E_BA_AC_OpMod01.eNightCooling]		:= TRUE;
	OuADmpOpMod.arrIgnoreDelayOffVal[E_BA_AC_OpMod01.eNightCooling]		:= TRUE;
	OuADmpOpMod.arrIgnoreFdbVal[E_BA_AC_OpMod01.eNightCooling]			:= FALSE;
	//////////////////////////////////////////////
	//////////////////////////////////////////////
	//	E_BA_AC_OpMod01.eCoolDownProtection;
	OuADmpOpMod.arrOpModVal[E_BA_AC_OpMod01.eCoolDownProtection]				:= TRUE;
	OuADmpOpMod.arrIgnoreDelayOnVal[E_BA_AC_OpMod01.eCoolDownProtection]		:= TRUE;
	OuADmpOpMod.arrIgnoreDelayOffVal[E_BA_AC_OpMod01.eCoolDownProtection]	:= TRUE;
	OuADmpOpMod.arrIgnoreFdbVal[E_BA_AC_OpMod01.eCoolDownProtection]			:= FALSE;
	//////////////////////////////////////////////
	//////////////////////////////////////////////
	//	E_BA_AC_OpMod01.eOverHeatingProtection;
	OuADmpOpMod.arrOpModVal[E_BA_AC_OpMod01.eOverHeatingProtection]				:= TRUE;
	OuADmpOpMod.arrIgnoreDelayOnVal[E_BA_AC_OpMod01.eOverHeatingProtection]		:= TRUE;
	OuADmpOpMod.arrIgnoreDelayOffVal[E_BA_AC_OpMod01.eOverHeatingProtection]		:= TRUE;
	OuADmpOpMod.arrIgnoreFdbVal[E_BA_AC_OpMod01.eOverHeatingProtection]			:= FALSE;
	//////////////////////////////////////////////
	//////////////////////////////////////////////
	//	E_BA_AC_OpMod01.eAlarm;
	OuADmpOpMod.arrOpModVal[E_BA_AC_OpMod01.eAlarm]				:= FALSE;
	OuADmpOpMod.arrIgnoreDelayOnVal[E_BA_AC_OpMod01.eAlarm]		:= TRUE;
	OuADmpOpMod.arrIgnoreDelayOffVal[E_BA_AC_OpMod01.eAlarm]		:= FALSE;
	OuADmpOpMod.arrIgnoreFdbVal[E_BA_AC_OpMod01.eAlarm]			:= TRUE;
	//////////////////////////////////////////////
	//////////////////////////////////////////////
	//	E_BA_AC_OpMod01.eForcedVentilation;
	OuADmpOpMod.arrOpModVal[E_BA_AC_OpMod01.eForcedVentilation]				:= TRUE;
	OuADmpOpMod.arrIgnoreDelayOnVal[E_BA_AC_OpMod01.eForcedVentilation]		:= TRUE;
	OuADmpOpMod.arrIgnoreDelayOffVal[E_BA_AC_OpMod01.eForcedVentilation]		:= TRUE;
	OuADmpOpMod.arrIgnoreFdbVal[E_BA_AC_OpMod01.eForcedVentilation]			:= FALSE;
	//////////////////////////////////////////////
	//////////////////////////////////////////////
	//	E_BA_AC_OpMod01.eCentralSwitchOff;
	OuADmpOpMod.arrOpModVal[E_BA_AC_OpMod01.eCentralSwitchOff]				:= FALSE;
	OuADmpOpMod.arrIgnoreDelayOnVal[E_BA_AC_OpMod01.eCentralSwitchOff]		:= TRUE;
	OuADmpOpMod.arrIgnoreDelayOffVal[E_BA_AC_OpMod01.eCentralSwitchOff]		:= FALSE;
	OuADmpOpMod.arrIgnoreFdbVal[E_BA_AC_OpMod01.eCentralSwitchOff]			:= TRUE;
	//////////////////////////////////////////////
	//////////////////////////////////////////////
	//	E_BA_AC_OpMod01.eCustomer01
	OuADmpOpMod.arrOpModVal[E_BA_AC_OpMod01.eCustomer01]				:= FALSE;
	OuADmpOpMod.arrIgnoreDelayOnVal[E_BA_AC_OpMod01.eCustomer01]		:= TRUE;
	OuADmpOpMod.arrIgnoreDelayOffVal[E_BA_AC_OpMod01.eCustomer01]	:= FALSE;
	OuADmpOpMod.arrIgnoreFdbVal[E_BA_AC_OpMod01.eCustomer01]			:= TRUE;
	//////////////////////////////////////////////
	//////////////////////////////////////////////
	//	E_BA_AC_OpMod01.eCustomer02
	OuADmpOpMod.arrOpModVal[E_BA_AC_OpMod01.eCustomer02]				:= FALSE;
	OuADmpOpMod.arrIgnoreDelayOnVal[E_BA_AC_OpMod01.eCustomer02]		:= TRUE;
	OuADmpOpMod.arrIgnoreDelayOffVal[E_BA_AC_OpMod01.eCustomer02]	:= FALSE;
	OuADmpOpMod.arrIgnoreFdbVal[E_BA_AC_OpMod01.eCustomer02]			:= TRUE;
END_IF
END_METHOD

METHOD InitPreHtr
VAR_INPUT
END_VAR
IF	PreHtrOpMod.bInit
THEN	
	PreHtrOpMod.bInit := FALSE;
	//////////////////////////////////////////////
	//////////////////////////////////////////////
	//	E_BA_AC_OpMod01.eOff;
	PreHtrOpMod.arrOpModVal[E_BA_AC_OpMod01.eOff]				:= FALSE;
	PreHtrOpMod.arrIgnoreDelayOnVal[E_BA_AC_OpMod01.eOff]		:= TRUE;
	PreHtrOpMod.arrIgnoreDelayOffVal[E_BA_AC_OpMod01.eOff]		:= TRUE;
	PreHtrOpMod.arrIgnoreFdbVal[E_BA_AC_OpMod01.eOff]			:= TRUE;
	//////////////////////////////////////////////
	//////////////////////////////////////////////
	//	E_BA_AC_OpMod01.eOn;
	PreHtrOpMod.arrOpModVal[E_BA_AC_OpMod01.eOn]				:= TRUE;
	PreHtrOpMod.arrIgnoreDelayOnVal[E_BA_AC_OpMod01.eOn]		:= TRUE;
	PreHtrOpMod.arrIgnoreDelayOffVal[E_BA_AC_OpMod01.eOn]	:= TRUE;
	PreHtrOpMod.arrIgnoreFdbVal[E_BA_AC_OpMod01.eOn]			:= FALSE;
	//////////////////////////////////////////////
	//////////////////////////////////////////////
	//	E_BA_AC_OpMod01.eEmergency;
	PreHtrOpMod.arrOpModVal[E_BA_AC_OpMod01.eEmergency]				:= FALSE;
	PreHtrOpMod.arrIgnoreDelayOnVal[E_BA_AC_OpMod01.eEmergency]		:= TRUE;
	PreHtrOpMod.arrIgnoreDelayOffVal[E_BA_AC_OpMod01.eEmergency]		:= TRUE;
	PreHtrOpMod.arrIgnoreFdbVal[E_BA_AC_OpMod01.eEmergency]			:= TRUE;
	//////////////////////////////////////////////
	//////////////////////////////////////////////
	//	E_BA_AC_OpMod01.eFrost;
	PreHtrOpMod.arrOpModVal[E_BA_AC_OpMod01.eFrost]				:= FALSE;
	PreHtrOpMod.arrIgnoreDelayOnVal[E_BA_AC_OpMod01.eFrost]		:= TRUE;
	PreHtrOpMod.arrIgnoreDelayOffVal[E_BA_AC_OpMod01.eFrost]		:= TRUE;
	PreHtrOpMod.arrIgnoreFdbVal[E_BA_AC_OpMod01.eFrost]			:= TRUE;
	//////////////////////////////////////////////
	//////////////////////////////////////////////
	//	E_BA_AC_OpMod01.eSmokeExtractionProgram;
	PreHtrOpMod.arrOpModVal[E_BA_AC_OpMod01.eSmokeExtractionProgram]				:= TRUE;
	PreHtrOpMod.arrIgnoreDelayOnVal[E_BA_AC_OpMod01.eSmokeExtractionProgram]		:= TRUE;
	PreHtrOpMod.arrIgnoreDelayOffVal[E_BA_AC_OpMod01.eSmokeExtractionProgram]	:= TRUE;
	PreHtrOpMod.arrIgnoreFdbVal[E_BA_AC_OpMod01.eSmokeExtractionProgram]			:= TRUE;
	//////////////////////////////////////////////
	//////////////////////////////////////////////
	//	E_BA_AC_OpMod01.eSmokeExtractionSupplyAir;
	PreHtrOpMod.arrOpModVal[E_BA_AC_OpMod01.eSmokeExtractionSupplyAir]				:= TRUE;
	PreHtrOpMod.arrIgnoreDelayOnVal[E_BA_AC_OpMod01.eSmokeExtractionSupplyAir]		:= TRUE;
	PreHtrOpMod.arrIgnoreDelayOffVal[E_BA_AC_OpMod01.eSmokeExtractionSupplyAir]		:= TRUE;
	PreHtrOpMod.arrIgnoreFdbVal[E_BA_AC_OpMod01.eSmokeExtractionSupplyAir]			:= TRUE;
	//////////////////////////////////////////////
	//////////////////////////////////////////////
	//	E_BA_AC_OpMod01.eSmokeExtractionExhaustAir;
	PreHtrOpMod.arrOpModVal[E_BA_AC_OpMod01.eSmokeExtractionExhaustAir]				:= FALSE;
	PreHtrOpMod.arrIgnoreDelayOnVal[E_BA_AC_OpMod01.eSmokeExtractionExhaustAir]		:= TRUE;
	PreHtrOpMod.arrIgnoreDelayOffVal[E_BA_AC_OpMod01.eSmokeExtractionExhaustAir]		:= TRUE;
	PreHtrOpMod.arrIgnoreFdbVal[E_BA_AC_OpMod01.eSmokeExtractionExhaustAir]			:= TRUE;
	//////////////////////////////////////////////
	//////////////////////////////////////////////
	//	E_BA_AC_OpMod01.eFire;
	PreHtrOpMod.arrOpModVal[E_BA_AC_OpMod01.eFire]				:= FALSE;
	PreHtrOpMod.arrIgnoreDelayOnVal[E_BA_AC_OpMod01.eFire]		:= TRUE;
	PreHtrOpMod.arrIgnoreDelayOffVal[E_BA_AC_OpMod01.eFire]		:= TRUE;
	PreHtrOpMod.arrIgnoreFdbVal[E_BA_AC_OpMod01.eFire]			:= TRUE;
	//////////////////////////////////////////////
	//////////////////////////////////////////////
	//	E_BA_AC_OpMod01.eNightCooling;
	PreHtrOpMod.arrOpModVal[E_BA_AC_OpMod01.eNightCooling]				:= FALSE;
	PreHtrOpMod.arrIgnoreDelayOnVal[E_BA_AC_OpMod01.eNightCooling]		:= TRUE;
	PreHtrOpMod.arrIgnoreDelayOffVal[E_BA_AC_OpMod01.eNightCooling]		:= TRUE;
	PreHtrOpMod.arrIgnoreFdbVal[E_BA_AC_OpMod01.eNightCooling]			:= TRUE;
	//////////////////////////////////////////////
	//////////////////////////////////////////////
	//	E_BA_AC_OpMod01.eCoolDownProtection;
	PreHtrOpMod.arrOpModVal[E_BA_AC_OpMod01.eCoolDownProtection]				:= TRUE;
	PreHtrOpMod.arrIgnoreDelayOnVal[E_BA_AC_OpMod01.eCoolDownProtection]		:= TRUE;
	PreHtrOpMod.arrIgnoreDelayOffVal[E_BA_AC_OpMod01.eCoolDownProtection]	:= TRUE;
	PreHtrOpMod.arrIgnoreFdbVal[E_BA_AC_OpMod01.eCoolDownProtection]			:= FALSE;
	//////////////////////////////////////////////
	//////////////////////////////////////////////
	//	E_BA_AC_OpMod01.eOverHeatingProtection;
	PreHtrOpMod.arrOpModVal[E_BA_AC_OpMod01.eOverHeatingProtection]				:= FALSE;
	PreHtrOpMod.arrIgnoreDelayOnVal[E_BA_AC_OpMod01.eOverHeatingProtection]		:= TRUE;
	PreHtrOpMod.arrIgnoreDelayOffVal[E_BA_AC_OpMod01.eOverHeatingProtection]		:= TRUE;
	PreHtrOpMod.arrIgnoreFdbVal[E_BA_AC_OpMod01.eOverHeatingProtection]			:= TRUE;
	//////////////////////////////////////////////
	//////////////////////////////////////////////
	//	E_BA_AC_OpMod01.eAlarm;
	PreHtrOpMod.arrOpModVal[E_BA_AC_OpMod01.eAlarm]				:= FALSE;
	PreHtrOpMod.arrIgnoreDelayOnVal[E_BA_AC_OpMod01.eAlarm]		:= TRUE;
	PreHtrOpMod.arrIgnoreDelayOffVal[E_BA_AC_OpMod01.eAlarm]		:= TRUE;
	PreHtrOpMod.arrIgnoreFdbVal[E_BA_AC_OpMod01.eAlarm]			:= TRUE;
	//////////////////////////////////////////////
	//////////////////////////////////////////////
	//	E_BA_AC_OpMod01.eForcedVentilation;
	PreHtrOpMod.arrOpModVal[E_BA_AC_OpMod01.eForcedVentilation]				:= TRUE;
	PreHtrOpMod.arrIgnoreDelayOnVal[E_BA_AC_OpMod01.eForcedVentilation]		:= TRUE;
	PreHtrOpMod.arrIgnoreDelayOffVal[E_BA_AC_OpMod01.eForcedVentilation]		:= TRUE;
	PreHtrOpMod.arrIgnoreFdbVal[E_BA_AC_OpMod01.eForcedVentilation]			:= FALSE;
	//////////////////////////////////////////////
	//////////////////////////////////////////////
	//	E_BA_AC_OpMod01.eCentralSwitchOff;
	PreHtrOpMod.arrOpModVal[E_BA_AC_OpMod01.eCentralSwitchOff]				:= FALSE;
	PreHtrOpMod.arrIgnoreDelayOnVal[E_BA_AC_OpMod01.eCentralSwitchOff]		:= TRUE;
	PreHtrOpMod.arrIgnoreDelayOffVal[E_BA_AC_OpMod01.eCentralSwitchOff]		:= TRUE;
	PreHtrOpMod.arrIgnoreFdbVal[E_BA_AC_OpMod01.eCentralSwitchOff]			:= TRUE;
	//////////////////////////////////////////////
	//////////////////////////////////////////////
	//	E_BA_AC_OpMod01.eCustomer01;
	PreHtrOpMod.arrOpModVal[E_BA_AC_OpMod01.eCustomer01]				:= FALSE;
	PreHtrOpMod.arrIgnoreDelayOnVal[E_BA_AC_OpMod01.eCustomer01]		:= TRUE;
	PreHtrOpMod.arrIgnoreDelayOffVal[E_BA_AC_OpMod01.eCustomer01]	:= TRUE;
	PreHtrOpMod.arrIgnoreFdbVal[E_BA_AC_OpMod01.eCustomer01]			:= TRUE;
	//////////////////////////////////////////////
	//////////////////////////////////////////////
	//	E_BA_AC_OpMod01.eCustomer02;
	PreHtrOpMod.arrOpModVal[E_BA_AC_OpMod01.eCustomer02]				:= FALSE;
	PreHtrOpMod.arrIgnoreDelayOnVal[E_BA_AC_OpMod01.eCustomer02]		:= TRUE;
	PreHtrOpMod.arrIgnoreDelayOffVal[E_BA_AC_OpMod01.eCustomer02]	:= TRUE;
	PreHtrOpMod.arrIgnoreFdbVal[E_BA_AC_OpMod01.eCustomer02]			:= TRUE;
END_IF
END_METHOD

METHOD InitSuAFan
VAR_INPUT
END_VAR
IF	SuAFanOpMod.bInit
THEN	
	SuAFanOpMod.bInit := FALSE;
	//////////////////////////////////////////////
	//////////////////////////////////////////////
	//	E_BA_AC_OpMod01.eOff;
	SuAFanOpMod.arrOpModVal[E_BA_AC_OpMod01.eOff]				:= E_BA_Mdlt.eOff;
	SuAFanOpMod.arrIgnoreDelayOnVal[E_BA_AC_OpMod01.eOff]		:= TRUE;
	SuAFanOpMod.arrIgnoreDelayOffVal[E_BA_AC_OpMod01.eOff]		:= FALSE;
	SuAFanOpMod.arrIgnoreFdbVal[E_BA_AC_OpMod01.eOff]			:= TRUE;
	//////////////////////////////////////////////
	//////////////////////////////////////////////
	//	E_BA_AC_OpMod01.eOn;
	SuAFanOpMod.arrOpModVal[E_BA_AC_OpMod01.eOn]				:= E_BA_Mdlt.eOn;
	SuAFanOpMod.arrIgnoreDelayOnVal[E_BA_AC_OpMod01.eOn]		:= FALSE;
	SuAFanOpMod.arrIgnoreDelayOffVal[E_BA_AC_OpMod01.eOn]	:= TRUE;
	SuAFanOpMod.arrIgnoreFdbVal[E_BA_AC_OpMod01.eOn]			:= TRUE;
	//////////////////////////////////////////////
	//////////////////////////////////////////////
	//	E_BA_AC_OpMod01.eEmergency;
	SuAFanOpMod.arrOpModVal[E_BA_AC_OpMod01.eEmergency]				:= E_BA_Mdlt.eOff;
	SuAFanOpMod.arrIgnoreDelayOnVal[E_BA_AC_OpMod01.eEmergency]		:= TRUE;
	SuAFanOpMod.arrIgnoreDelayOffVal[E_BA_AC_OpMod01.eEmergency]		:= FALSE;
	SuAFanOpMod.arrIgnoreFdbVal[E_BA_AC_OpMod01.eEmergency]			:= TRUE;
	//////////////////////////////////////////////
	//////////////////////////////////////////////
	//	E_BA_AC_OpMod01.eFrost;
	SuAFanOpMod.arrOpModVal[E_BA_AC_OpMod01.eFrost]				:= E_BA_Mdlt.eOff;
	SuAFanOpMod.arrIgnoreDelayOnVal[E_BA_AC_OpMod01.eFrost]		:= TRUE;
	SuAFanOpMod.arrIgnoreDelayOffVal[E_BA_AC_OpMod01.eFrost]		:= FALSE;
	SuAFanOpMod.arrIgnoreFdbVal[E_BA_AC_OpMod01.eFrost]			:= TRUE;
	//////////////////////////////////////////////
	//////////////////////////////////////////////
	//	E_BA_AC_OpMod01.eSmokeExtractionProgram;
	SuAFanOpMod.arrOpModVal[E_BA_AC_OpMod01.eSmokeExtractionProgram]				:= E_BA_Mdlt.eOn;
	SuAFanOpMod.arrIgnoreDelayOnVal[E_BA_AC_OpMod01.eSmokeExtractionProgram]		:= TRUE;
	SuAFanOpMod.arrIgnoreDelayOffVal[E_BA_AC_OpMod01.eSmokeExtractionProgram]		:= FALSE;
	SuAFanOpMod.arrIgnoreFdbVal[E_BA_AC_OpMod01.eSmokeExtractionProgram]			:= TRUE;
	//////////////////////////////////////////////
	//////////////////////////////////////////////
	//	E_BA_AC_OpMod01.eSmokeExtractionSupplyAir;
	SuAFanOpMod.arrOpModVal[E_BA_AC_OpMod01.eSmokeExtractionSupplyAir]				:= E_BA_Mdlt.eOn;
	SuAFanOpMod.arrIgnoreDelayOnVal[E_BA_AC_OpMod01.eSmokeExtractionSupplyAir]		:= TRUE;
	SuAFanOpMod.arrIgnoreDelayOffVal[E_BA_AC_OpMod01.eSmokeExtractionSupplyAir]		:= TRUE;
	SuAFanOpMod.arrIgnoreFdbVal[E_BA_AC_OpMod01.eSmokeExtractionSupplyAir]			:= TRUE;
	//////////////////////////////////////////////
	//////////////////////////////////////////////
	//	E_BA_AC_OpMod01.eSmokeExtractionExhaustAir;
	SuAFanOpMod.arrOpModVal[E_BA_AC_OpMod01.eSmokeExtractionExhaustAir]				:= E_BA_Mdlt.eOff;
	SuAFanOpMod.arrIgnoreDelayOnVal[E_BA_AC_OpMod01.eSmokeExtractionExhaustAir]		:= TRUE;
	SuAFanOpMod.arrIgnoreDelayOffVal[E_BA_AC_OpMod01.eSmokeExtractionExhaustAir]		:= FALSE;
	SuAFanOpMod.arrIgnoreFdbVal[E_BA_AC_OpMod01.eSmokeExtractionExhaustAir]			:= TRUE;
	//////////////////////////////////////////////
	//////////////////////////////////////////////
	//	E_BA_AC_OpMod01.eFire;
	SuAFanOpMod.arrOpModVal[E_BA_AC_OpMod01.eFire]				:= E_BA_Mdlt.eOff;
	SuAFanOpMod.arrIgnoreDelayOnVal[E_BA_AC_OpMod01.eFire]		:= TRUE;
	SuAFanOpMod.arrIgnoreDelayOffVal[E_BA_AC_OpMod01.eFire]		:= FALSE;
	SuAFanOpMod.arrIgnoreFdbVal[E_BA_AC_OpMod01.eFire]			:= TRUE;
	//////////////////////////////////////////////
	//////////////////////////////////////////////
	//	E_BA_AC_OpMod01.eNightCooling;
	SuAFanOpMod.arrOpModVal[E_BA_AC_OpMod01.eNightCooling]				:= E_BA_Mdlt.eOn;
	SuAFanOpMod.arrIgnoreDelayOnVal[E_BA_AC_OpMod01.eNightCooling]		:= FALSE;
	SuAFanOpMod.arrIgnoreDelayOffVal[E_BA_AC_OpMod01.eNightCooling]		:= TRUE;
	SuAFanOpMod.arrIgnoreFdbVal[E_BA_AC_OpMod01.eNightCooling]			:= TRUE;
	//////////////////////////////////////////////
	//////////////////////////////////////////////
	//	E_BA_AC_OpMod01.eCoolDownProtection;
	SuAFanOpMod.arrOpModVal[E_BA_AC_OpMod01.eCoolDownProtection]				:= E_BA_Mdlt.eOn;
	SuAFanOpMod.arrIgnoreDelayOnVal[E_BA_AC_OpMod01.eCoolDownProtection]		:= FALSE;
	SuAFanOpMod.arrIgnoreDelayOffVal[E_BA_AC_OpMod01.eCoolDownProtection]	:= TRUE;
	SuAFanOpMod.arrIgnoreFdbVal[E_BA_AC_OpMod01.eCoolDownProtection]			:= TRUE;
	//////////////////////////////////////////////
	//////////////////////////////////////////////
	//	E_BA_AC_OpMod01.eOverHeatingProtection;
	SuAFanOpMod.arrOpModVal[E_BA_AC_OpMod01.eOverHeatingProtection]				:= E_BA_Mdlt.eOn;
	SuAFanOpMod.arrIgnoreDelayOnVal[E_BA_AC_OpMod01.eOverHeatingProtection]		:= FALSE;
	SuAFanOpMod.arrIgnoreDelayOffVal[E_BA_AC_OpMod01.eOverHeatingProtection]		:= TRUE;
	SuAFanOpMod.arrIgnoreFdbVal[E_BA_AC_OpMod01.eOverHeatingProtection]			:= TRUE;
	//////////////////////////////////////////////
	//////////////////////////////////////////////
	//	E_BA_AC_OpMod01.eAlarm;
	SuAFanOpMod.arrOpModVal[E_BA_AC_OpMod01.eAlarm]				:= E_BA_Mdlt.eOff;
	SuAFanOpMod.arrIgnoreDelayOnVal[E_BA_AC_OpMod01.eAlarm]		:= TRUE;
	SuAFanOpMod.arrIgnoreDelayOffVal[E_BA_AC_OpMod01.eAlarm]		:= FALSE;
	SuAFanOpMod.arrIgnoreFdbVal[E_BA_AC_OpMod01.eAlarm]			:= TRUE;
	//////////////////////////////////////////////
	//////////////////////////////////////////////
	//	E_BA_AC_OpMod01.eForcedVentilation;
	SuAFanOpMod.arrOpModVal[E_BA_AC_OpMod01.eForcedVentilation]				:= E_BA_Mdlt.eOn;
	SuAFanOpMod.arrIgnoreDelayOnVal[E_BA_AC_OpMod01.eForcedVentilation]		:= TRUE;
	SuAFanOpMod.arrIgnoreDelayOffVal[E_BA_AC_OpMod01.eForcedVentilation]		:= TRUE;
	SuAFanOpMod.arrIgnoreFdbVal[E_BA_AC_OpMod01.eForcedVentilation]			:= TRUE;
	//////////////////////////////////////////////
	//////////////////////////////////////////////
	//	E_BA_AC_OpMod01.eCentralSwitchOff;
	SuAFanOpMod.arrOpModVal[E_BA_AC_OpMod01.eCentralSwitchOff]				:= E_BA_Mdlt.eOff;
	SuAFanOpMod.arrIgnoreDelayOnVal[E_BA_AC_OpMod01.eCentralSwitchOff]		:= TRUE;
	SuAFanOpMod.arrIgnoreDelayOffVal[E_BA_AC_OpMod01.eCentralSwitchOff]		:= FALSE;
	SuAFanOpMod.arrIgnoreFdbVal[E_BA_AC_OpMod01.eCentralSwitchOff]			:= TRUE;
	//////////////////////////////////////////////
	//////////////////////////////////////////////
	//	E_BA_AC_OpMod01.eCustomer01;
	SuAFanOpMod.arrOpModVal[E_BA_AC_OpMod01.eCustomer01]				:= E_BA_Mdlt.eOff;
	SuAFanOpMod.arrIgnoreDelayOnVal[E_BA_AC_OpMod01.eCustomer01]		:= TRUE;
	SuAFanOpMod.arrIgnoreDelayOffVal[E_BA_AC_OpMod01.eCustomer01]	:= FALSE;
	SuAFanOpMod.arrIgnoreFdbVal[E_BA_AC_OpMod01.eCustomer01]			:= TRUE;
	//////////////////////////////////////////////
	//////////////////////////////////////////////
	//	E_BA_AC_OpMod01.eCustomer02;
	SuAFanOpMod.arrOpModVal[E_BA_AC_OpMod01.eCustomer02]				:= E_BA_Mdlt.eOff;
	SuAFanOpMod.arrIgnoreDelayOnVal[E_BA_AC_OpMod01.eCustomer02]		:= TRUE;
	SuAFanOpMod.arrIgnoreDelayOffVal[E_BA_AC_OpMod01.eCustomer02]	:= FALSE;
	SuAFanOpMod.arrIgnoreFdbVal[E_BA_AC_OpMod01.eCustomer02]			:= TRUE;
END_IF
END_METHOD

METHOD InitTempCtrl
VAR_INPUT
END_VAR
IF	TempCtrlOpMod.bInit
THEN	
	TempCtrlOpMod.bInit := FALSE;
	//////////////////////////////////////////////
	//////////////////////////////////////////////
	//	E_BA_AC_OpMod01.eOff;
	TempCtrlOpMod.arrOpModVal[E_BA_AC_OpMod01.eOff]					:= E_BA_Mdlt.eOff;
	TempCtrlOpMod.arrIgnoreDelayOnVal[E_BA_AC_OpMod01.eOff]			:= TRUE;
	TempCtrlOpMod.arrIgnoreDelayOffVal[E_BA_AC_OpMod01.eOff]			:= TRUE;
	TempCtrlOpMod.arrIgnoreFdbVal[E_BA_AC_OpMod01.eOff]				:= TRUE;
	//////////////////////////////////////////////
	//////////////////////////////////////////////
	//	E_BA_AC_OpMod01.eOn;
	TempCtrlOpMod.arrOpModVal[E_BA_AC_OpMod01.eOn]					:= E_BA_Mdlt.eOn;
	TempCtrlOpMod.arrIgnoreDelayOnVal[E_BA_AC_OpMod01.eOn]			:= FALSE;
	TempCtrlOpMod.arrIgnoreDelayOffVal[E_BA_AC_OpMod01.eOn]			:= TRUE;
	TempCtrlOpMod.arrIgnoreFdbVal[E_BA_AC_OpMod01.eOn]				:= TRUE;
	//////////////////////////////////////////////
	//////////////////////////////////////////////
	//	E_BA_AC_OpMod01.eEmergency;	
	TempCtrlOpMod.arrOpModVal[E_BA_AC_OpMod01.eEmergency]					:= E_BA_Mdlt.eOff;
	TempCtrlOpMod.arrIgnoreDelayOnVal[E_BA_AC_OpMod01.eEmergency]			:= TRUE;
	TempCtrlOpMod.arrIgnoreDelayOffVal[E_BA_AC_OpMod01.eEmergency]			:= TRUE;
	TempCtrlOpMod.arrIgnoreFdbVal[E_BA_AC_OpMod01.eEmergency]				:= TRUE;
	//////////////////////////////////////////////
	//////////////////////////////////////////////
	//	E_BA_AC_OpMod01.eFrost;
	TempCtrlOpMod.arrOpModVal[E_BA_AC_OpMod01.eFrost]					:= E_BA_Mdlt.eOff;
	TempCtrlOpMod.arrIgnoreDelayOnVal[E_BA_AC_OpMod01.eFrost]			:= TRUE;
	TempCtrlOpMod.arrIgnoreDelayOffVal[E_BA_AC_OpMod01.eFrost]			:= TRUE;
	TempCtrlOpMod.arrIgnoreFdbVal[E_BA_AC_OpMod01.eFrost]				:= TRUE;
	//////////////////////////////////////////////
	//////////////////////////////////////////////
	//	E_BA_AC_OpMod01.eSmokeExtractionProgram;
	TempCtrlOpMod.arrOpModVal[E_BA_AC_OpMod01.eSmokeExtractionProgram]					:= E_BA_Mdlt.eOn;
	TempCtrlOpMod.arrIgnoreDelayOnVal[E_BA_AC_OpMod01.eSmokeExtractionProgram]			:= TRUE;
	TempCtrlOpMod.arrIgnoreDelayOffVal[E_BA_AC_OpMod01.eSmokeExtractionProgram]			:= TRUE;
	TempCtrlOpMod.arrIgnoreFdbVal[E_BA_AC_OpMod01.eSmokeExtractionProgram]				:= TRUE;
	//////////////////////////////////////////////
	//////////////////////////////////////////////
	//	E_BA_AC_OpMod01.eSmokeExtractionSupplyAir;
	TempCtrlOpMod.arrOpModVal[E_BA_AC_OpMod01.eSmokeExtractionSupplyAir]					:= E_BA_Mdlt.eOn; 
	TempCtrlOpMod.arrIgnoreDelayOnVal[E_BA_AC_OpMod01.eSmokeExtractionSupplyAir]			:= TRUE; 
	TempCtrlOpMod.arrIgnoreDelayOffVal[E_BA_AC_OpMod01.eSmokeExtractionSupplyAir]			:= TRUE; 
	TempCtrlOpMod.arrIgnoreFdbVal[E_BA_AC_OpMod01.eSmokeExtractionSupplyAir]				:= TRUE; 
	//////////////////////////////////////////////
	//////////////////////////////////////////////
	//	E_BA_AC_OpMod01.eSmokeExtractionExhaustAir;
	TempCtrlOpMod.arrOpModVal[E_BA_AC_OpMod01.eSmokeExtractionExhaustAir]					:= E_BA_Mdlt.eOn; 
	TempCtrlOpMod.arrIgnoreDelayOnVal[E_BA_AC_OpMod01.eSmokeExtractionExhaustAir]			:= TRUE; 
	TempCtrlOpMod.arrIgnoreDelayOffVal[E_BA_AC_OpMod01.eSmokeExtractionExhaustAir]			:= TRUE; 
	TempCtrlOpMod.arrIgnoreFdbVal[E_BA_AC_OpMod01.eSmokeExtractionExhaustAir]				:= TRUE; 
	//////////////////////////////////////////////
	//////////////////////////////////////////////
	//	E_BA_AC_OpMod01.eFire;
	TempCtrlOpMod.arrOpModVal[E_BA_AC_OpMod01.eFire]					:= E_BA_Mdlt.eOff; 
	TempCtrlOpMod.arrIgnoreDelayOnVal[E_BA_AC_OpMod01.eFire]			:= TRUE; 
	TempCtrlOpMod.arrIgnoreDelayOffVal[E_BA_AC_OpMod01.eFire]			:= TRUE; 
	TempCtrlOpMod.arrIgnoreFdbVal[E_BA_AC_OpMod01.eFire]				:= TRUE; 
	//////////////////////////////////////////////
	//////////////////////////////////////////////
	//	E_BA_AC_OpMod01.eNightCooling;
	TempCtrlOpMod.arrOpModVal[E_BA_AC_OpMod01.eNightCooling]					:= E_BA_Mdlt.eOn; 
	TempCtrlOpMod.arrIgnoreDelayOnVal[E_BA_AC_OpMod01.eNightCooling]			:= FALSE; 
	TempCtrlOpMod.arrIgnoreDelayOffVal[E_BA_AC_OpMod01.eNightCooling]			:= TRUE; 
	TempCtrlOpMod.arrIgnoreFdbVal[E_BA_AC_OpMod01.eNightCooling]				:= TRUE; 
	//////////////////////////////////////////////
	//////////////////////////////////////////////
	//	E_BA_AC_OpMod01.eCoolDownProtection;
	TempCtrlOpMod.arrOpModVal[E_BA_AC_OpMod01.eCoolDownProtection]				:= E_BA_Mdlt.eMax; 
	TempCtrlOpMod.arrIgnoreDelayOnVal[E_BA_AC_OpMod01.eCoolDownProtection]		:= FALSE; 
	TempCtrlOpMod.arrIgnoreDelayOffVal[E_BA_AC_OpMod01.eCoolDownProtection]		:= TRUE; 
	TempCtrlOpMod.arrIgnoreFdbVal[E_BA_AC_OpMod01.eCoolDownProtection]			:= TRUE; 
	//////////////////////////////////////////////
	//////////////////////////////////////////////
	//	E_BA_AC_OpMod01.eOverHeatingProtection;
	TempCtrlOpMod.arrOpModVal[E_BA_AC_OpMod01.eOverHeatingProtection]				:= E_BA_Mdlt.eOn; 
	TempCtrlOpMod.arrIgnoreDelayOnVal[E_BA_AC_OpMod01.eOverHeatingProtection]		:= FALSE; 
	TempCtrlOpMod.arrIgnoreDelayOffVal[E_BA_AC_OpMod01.eOverHeatingProtection]		:= TRUE; 
	TempCtrlOpMod.arrIgnoreFdbVal[E_BA_AC_OpMod01.eOverHeatingProtection]			:= TRUE; 
	//////////////////////////////////////////////
	//////////////////////////////////////////////
	//	E_BA_AC_OpMod01.eAlarm;
	TempCtrlOpMod.arrOpModVal[E_BA_AC_OpMod01.eAlarm]				:= E_BA_Mdlt.eOff;
	TempCtrlOpMod.arrIgnoreDelayOnVal[E_BA_AC_OpMod01.eAlarm]		:= TRUE;
	TempCtrlOpMod.arrIgnoreDelayOffVal[E_BA_AC_OpMod01.eAlarm]		:= TRUE;
	TempCtrlOpMod.arrIgnoreFdbVal[E_BA_AC_OpMod01.eAlarm]			:= TRUE;
	//////////////////////////////////////////////
	//////////////////////////////////////////////
	//	E_BA_AC_OpMod01.eForcedVentilation;
	TempCtrlOpMod.arrOpModVal[E_BA_AC_OpMod01.eForcedVentilation]				:= E_BA_Mdlt.eOn;
	TempCtrlOpMod.arrIgnoreDelayOnVal[E_BA_AC_OpMod01.eForcedVentilation]		:= FALSE;
	TempCtrlOpMod.arrIgnoreDelayOffVal[E_BA_AC_OpMod01.eForcedVentilation]		:= TRUE;
	TempCtrlOpMod.arrIgnoreFdbVal[E_BA_AC_OpMod01.eForcedVentilation]			:= TRUE;
	//////////////////////////////////////////////
	//////////////////////////////////////////////
	//	E_BA_AC_OpMod01.eCentralSwitchOff;  	
	TempCtrlOpMod.arrOpModVal[E_BA_AC_OpMod01.eCentralSwitchOff]				:= E_BA_Mdlt.eOff;
	TempCtrlOpMod.arrIgnoreDelayOnVal[E_BA_AC_OpMod01.eCentralSwitchOff]		:= TRUE;
	TempCtrlOpMod.arrIgnoreDelayOffVal[E_BA_AC_OpMod01.eCentralSwitchOff]		:= TRUE;
	TempCtrlOpMod.arrIgnoreFdbVal[E_BA_AC_OpMod01.eCentralSwitchOff]			:= TRUE;
	//////////////////////////////////////////////
	//////////////////////////////////////////////
	//	E_BA_AC_OpMod01.eCustomer01
	TempCtrlOpMod.arrOpModVal[E_BA_AC_OpMod01.eCustomer01]				:= E_BA_Mdlt.eOff;
	TempCtrlOpMod.arrIgnoreDelayOnVal[E_BA_AC_OpMod01.eCustomer01]		:= TRUE;
	TempCtrlOpMod.arrIgnoreDelayOffVal[E_BA_AC_OpMod01.eCustomer01]		:= TRUE;
	TempCtrlOpMod.arrIgnoreFdbVal[E_BA_AC_OpMod01.eCustomer01]			:= TRUE;
	//////////////////////////////////////////////
	//////////////////////////////////////////////
	//	E_BA_AC_OpMod01.eCustomer02          	
	TempCtrlOpMod.arrOpModVal[E_BA_AC_OpMod01.eCustomer02]				:= E_BA_Mdlt.eOff;
	TempCtrlOpMod.arrIgnoreDelayOnVal[E_BA_AC_OpMod01.eCustomer02]		:= TRUE;
	TempCtrlOpMod.arrIgnoreDelayOffVal[E_BA_AC_OpMod01.eCustomer02]		:= TRUE;
	TempCtrlOpMod.arrIgnoreFdbVal[E_BA_AC_OpMod01.eCustomer02]			:= TRUE;
END_IF
END_METHOD

END_FUNCTION_BLOCK

(* stored: Version 1.1.0.1, ProductVersion 3.1.4024.12
   POU FB_BA_AC_PlantCmd_AHU_1st_10: Id {20345e30-8747-4d30-a7e1-1017ffd99d87}, SpecialFunc None
   Method CallInit: Id {9e03986c-d1e0-404b-9850-67dac4cf5f08}
   Method FB_init: Id {c0a6bb27-f646-44e7-a5fc-3672b82d5c2e}
   Method InitCooler: Id {e72e16f2-6364-4fac-8a14-70f922c35705}
   Method InitErc: Id {c209dd23-0c3c-44aa-9439-880ca1e7d9a7}
   Method InitExhADmp: Id {d3c5736b-5675-4f25-aef0-a152f82fde5d}
   Method InitExtAFan: Id {0003855f-e8a2-4581-aeb8-5599764c6e7c}
   Method InitOuADmp: Id {268261d8-ba06-4184-8573-487bc9aff2ea}
   Method InitPreHtr: Id {813643ab-b480-4fe6-8296-ff82cfdf4861}
   Method InitSuAFan: Id {96aa6dbe-c021-49e7-bdd8-9df194925230}
   Method InitTempCtrl: Id {61107a4a-3a81-4783-859a-1613cde2be15} *)
